  PROC DrawPart220()
    MoveL Offs(pOrigin,226.14,210.19,0.00),v60,z0,tPen\WObj:=wPaper;
    MoveL Offs(pOrigin,227.79,208.54,0.00),v40,fine,tPen\WObj:=wPaper;
    MoveL Offs(pOrigin,227.79,208.54,6.00),v60,z5,tPen\WObj:=wPaper;
    MoveL Offs(pOrigin,229.18,204.08,6.00),vTravel,z5,tPen\WObj:=wPaper;
    MoveL Offs(pOrigin,229.18,204.08,0.00),v60,z0,tPen\WObj:=wPaper;
    MoveL Offs(pOrigin,226.47,201.38,0.00),v40,fine,tPen\WObj:=wPaper;
    MoveL Offs(pOrigin,226.47,201.38,6.00),v60,z5,tPen\WObj:=wPaper;
    MoveL Offs(pOrigin,223.02,201.36,6.00),vTravel,z5,tPen\WObj:=wPaper;
    MoveL Offs(pOrigin,223.02,201.36,0.00),v60,z0,tPen\WObj:=wPaper;
    MoveL Offs(pOrigin,219.26,205.12,0.00),v40,fine,tPen\WObj:=wPaper;
    MoveL Offs(pOrigin,219.26,205.12,6.00),v60,z5,tPen\WObj:=wPaper;
    MoveL Offs(pOrigin,220.18,199.72,6.00),vTravel,z5,tPen\WObj:=wPaper;
    MoveL Offs(pOrigin,220.18,199.72,0.00),v60,z0,tPen\WObj:=wPaper;
    MoveL Offs(pOrigin,224.23,195.66,0.00),v40,fine,tPen\WObj:=wPaper;
    MoveL Offs(pOrigin,224.23,195.66,6.00),v60,z5,tPen\WObj:=wPaper;
    MoveL Offs(pOrigin,224.69,193.71,6.00),vTravel,z5,tPen\WObj:=wPaper;
    MoveL Offs(pOrigin,224.69,193.71,0.00),v60,z0,tPen\WObj:=wPaper;
    MoveL Offs(pOrigin,220.63,197.77,0.00),v40,fine,tPen\WObj:=wPaper;
    MoveL Offs(pOrigin,220.63,197.77,6.00),v60,z5,tPen\WObj:=wPaper;
    MoveL Offs(pOrigin,221.31,199.80,6.00),vTravel,z5,tPen\WObj:=wPaper;
    MoveL Offs(pOrigin,221.31,199.80,0.00),v60,z0,tPen\WObj:=wPaper;
    MoveL Offs(pOrigin,222.38,199.80,0.00),v40,fine,tPen\WObj:=wPaper;
    MoveL Offs(pOrigin,222.38,199.80,6.00),v60,z5,tPen\WObj:=wPaper;
    MoveL Offs(pOrigin,219.89,195.53,6.00),vTravel,z5,tPen\WObj:=wPaper;
    MoveL Offs(pOrigin,219.89,195.53,0.00),v60,z0,tPen\WObj:=wPaper;
    MoveL Offs(pOrigin,225.75,189.67,0.00),v40,fine,tPen\WObj:=wPaper;
    MoveL Offs(pOrigin,225.75,189.67,6.00),v60,z5,tPen\WObj:=wPaper;
    MoveL Offs(pOrigin,228.60,186.81,6.00),vTravel,z5,tPen\WObj:=wPaper;
    MoveL Offs(pOrigin,228.60,186.81,0.00),v60,z0,tPen\WObj:=wPaper;
    MoveL Offs(pOrigin,231.01,184.41,0.00),v40,z0,tPen\WObj:=wPaper;
    MoveL Offs(pOrigin,230.32,184.31,0.00),v40,z0,tPen\WObj:=wPaper;
    MoveL Offs(pOrigin,228.21,182.21,0.00),v40,fine,tPen\WObj:=wPaper;
    MoveL Offs(pOrigin,228.21,182.21,6.00),v60,z5,tPen\WObj:=wPaper;
    MoveL Offs(pOrigin,226.72,182.21,6.00),vTravel,z5,tPen\WObj:=wPaper;
    MoveL Offs(pOrigin,226.72,182.21,0.00),v60,z0,tPen\WObj:=wPaper;
    MoveL Offs(pOrigin,224.76,180.25,0.00),v40,z0,tPen\WObj:=wPaper;
    MoveL Offs(pOrigin,224.28,180.68,0.00),v40,z0,tPen\WObj:=wPaper;
    MoveL Offs(pOrigin,230.29,174.67,0.00),v40,z0,tPen\WObj:=wPaper;
    MoveL Offs(pOrigin,229.84,173.63,0.00),v40,z0,tPen\WObj:=wPaper;
    MoveL Offs(pOrigin,224.43,179.04,0.00),v40,z0,tPen\WObj:=wPaper;
    MoveL Offs(pOrigin,224.91,178.91,0.00),v40,z0,tPen\WObj:=wPaper;
    MoveL Offs(pOrigin,226.86,180.86,0.00),v40,z0,tPen\WObj:=wPaper;
    MoveL Offs(pOrigin,226.41,180.79,0.00),v40,z0,tPen\WObj:=wPaper;
    MoveL Offs(pOrigin,225.14,180.79,0.00),v40,z0,tPen\WObj:=wPaper;
    MoveL Offs(pOrigin,224.62,181.60,0.00),v40,z0,tPen\WObj:=wPaper;
    MoveL Offs(pOrigin,226.42,183.40,0.00),v40,z0,tPen\WObj:=wPaper;
    MoveL Offs(pOrigin,225.99,182.90,0.00),v40,z0,tPen\WObj:=wPaper;
    MoveL Offs(pOrigin,224.92,182.90,0.00),v40,z0,tPen\WObj:=wPaper;
    MoveL Offs(pOrigin,224.71,183.96,0.00),v40,z0,tPen\WObj:=wPaper;
    MoveL Offs(pOrigin,225.78,183.96,0.00),v40,fine,tPen\WObj:=wPaper;
    MoveL Offs(pOrigin,225.78,183.96,6.00),v60,z5,tPen\WObj:=wPaper;
    MoveL Offs(pOrigin,226.20,181.85,6.00),vTravel,z5,tPen\WObj:=wPaper;
    MoveL Offs(pOrigin,226.20,181.85,0.00),v60,z0,tPen\WObj:=wPaper;
    MoveL Offs(pOrigin,225.14,181.85,0.00),v40,fine,tPen\WObj:=wPaper;
    MoveL Offs(pOrigin,225.14,181.85,6.00),v60,z5,tPen\WObj:=wPaper;
    MoveL Offs(pOrigin,225.35,179.74,6.00),vTravel,z5,tPen\WObj:=wPaper;
    MoveL Offs(pOrigin,225.35,179.74,0.00),v60,z0,tPen\WObj:=wPaper;
    MoveL Offs(pOrigin,226.62,179.74,0.00),v40,z0,tPen\WObj:=wPaper;
    MoveL Offs(pOrigin,226.84,178.68,0.00),v40,z0,tPen\WObj:=wPaper;
    MoveL Offs(pOrigin,225.56,178.68,0.00),v40,fine,tPen\WObj:=wPaper;
    MoveL Offs(pOrigin,225.56,178.68,6.00),v60,z5,tPen\WObj:=wPaper;
    MoveL Offs(pOrigin,226.20,174.46,6.00),vTravel,z5,tPen\WObj:=wPaper;
    MoveL Offs(pOrigin,226.20,174.46,0.00),v60,z0,tPen\WObj:=wPaper;
    MoveL Offs(pOrigin,228.96,174.46,0.00),v40,fine,tPen\WObj:=wPaper;
    MoveL Offs(pOrigin,228.96,174.46,6.00),v60,z5,tPen\WObj:=wPaper;
    MoveL Offs(pOrigin,234.06,174.15,6.00),vTravel,z5,tPen\WObj:=wPaper;
    MoveL Offs(pOrigin,234.06,174.15,0.00),v60,z0,tPen\WObj:=wPaper;
    MoveL Offs(pOrigin,233.64,174.57,0.00),v40,z0,tPen\WObj:=wPaper;
    MoveL Offs(pOrigin,234.06,174.15,0.00),v40,fine,tPen\WObj:=wPaper;
    MoveL Offs(pOrigin,234.06,174.15,6.00),v60,z5,tPen\WObj:=wPaper;
    MoveL Offs(pOrigin,242.72,174.32,6.00),vTravel,z5,tPen\WObj:=wPaper;
    MoveL Offs(pOrigin,242.72,174.32,0.00),v60,z0,tPen\WObj:=wPaper;
    MoveL Offs(pOrigin,244.22,175.82,0.00),v40,fine,tPen\WObj:=wPaper;
    MoveL Offs(pOrigin,244.22,175.82,6.00),v60,z5,tPen\WObj:=wPaper;
    MoveL Offs(pOrigin,245.11,173.72,6.00),vTravel,z5,tPen\WObj:=wPaper;
    MoveL Offs(pOrigin,245.11,173.72,0.00),v60,z0,tPen\WObj:=wPaper;
    MoveL Offs(pOrigin,243.31,171.92,0.00),v40,fine,tPen\WObj:=wPaper;
    MoveL Offs(pOrigin,243.31,171.92,6.00),v60,z5,tPen\WObj:=wPaper;
    MoveL Offs(pOrigin,244.69,170.23,6.00),vTravel,z5,tPen\WObj:=wPaper;
    MoveL Offs(pOrigin,244.69,170.23,0.00),v60,z0,tPen\WObj:=wPaper;
    MoveL Offs(pOrigin,245.75,170.23,0.00),v40,z0,tPen\WObj:=wPaper;
    MoveL Offs(pOrigin,245.54,170.75,0.00),v40,z0,tPen\WObj:=wPaper;
    MoveL Offs(pOrigin,245.32,171.18,0.00),v40,z0,tPen\WObj:=wPaper;
    MoveL Offs(pOrigin,245.54,170.75,0.00),v40,z0,tPen\WObj:=wPaper;
    MoveL Offs(pOrigin,245.71,171.33,0.00),v40,z0,tPen\WObj:=wPaper;
    MoveL Offs(pOrigin,244.35,169.98,0.00),v40,z0,tPen\WObj:=wPaper;
    MoveL Offs(pOrigin,244.69,169.90,0.00),v40,z0,tPen\WObj:=wPaper;
    MoveL Offs(pOrigin,244.26,170.54,0.00),v40,z0,tPen\WObj:=wPaper;
    MoveL Offs(pOrigin,244.69,169.90,0.00),v40,z0,tPen\WObj:=wPaper;
    MoveL Offs(pOrigin,244.95,169.08,0.00),v40,z0,tPen\WObj:=wPaper;
    MoveL Offs(pOrigin,246.30,170.43,0.00),v40,z0,tPen\WObj:=wPaper;
    MoveL Offs(pOrigin,247.20,169.84,0.00),v40,z0,tPen\WObj:=wPaper;
    MoveL Offs(pOrigin,245.70,168.33,0.00),v40,z0,tPen\WObj:=wPaper;
    MoveL Offs(pOrigin,245.96,168.41,0.00),v40,z0,tPen\WObj:=wPaper;
    MoveL Offs(pOrigin,245.32,169.05,0.00),v40,z0,tPen\WObj:=wPaper;
    MoveL Offs(pOrigin,245.96,168.41,0.00),v40,z0,tPen\WObj:=wPaper;
    MoveL Offs(pOrigin,245.54,169.18,0.00),v40,z0,tPen\WObj:=wPaper;
    MoveL Offs(pOrigin,246.81,169.18,0.00),v40,z0,tPen\WObj:=wPaper;
    MoveL Offs(pOrigin,246.81,169.26,0.00),v40,z0,tPen\WObj:=wPaper;
    MoveL Offs(pOrigin,245.75,170.32,0.00),v40,z0,tPen\WObj:=wPaper;
    MoveL Offs(pOrigin,246.81,169.26,0.00),v40,fine,tPen\WObj:=wPaper;
    MoveL Offs(pOrigin,246.81,169.26,6.00),v60,z5,tPen\WObj:=wPaper;
    MoveL Offs(pOrigin,241.29,179.04,6.00),vTravel,z5,tPen\WObj:=wPaper;
    MoveL Offs(pOrigin,241.29,179.04,0.00),v60,z0,tPen\WObj:=wPaper;
    MoveL Offs(pOrigin,241.07,179.46,0.00),v40,z0,tPen\WObj:=wPaper;
    MoveL Offs(pOrigin,241.29,179.04,0.00),v40,z0,tPen\WObj:=wPaper;
    MoveL Offs(pOrigin,241.08,179.74,0.00),v40,z0,tPen\WObj:=wPaper;
    MoveL Offs(pOrigin,242.35,179.74,0.00),v40,fine,tPen\WObj:=wPaper;
    MoveL Offs(pOrigin,242.35,179.74,6.00),v60,z5,tPen\WObj:=wPaper;
    MoveL Offs(pOrigin,240.44,180.74,6.00),vTravel,z5,tPen\WObj:=wPaper;
    MoveL Offs(pOrigin,240.44,180.74,0.00),v60,z0,tPen\WObj:=wPaper;
    MoveL Offs(pOrigin,240.23,181.16,0.00),v40,z0,tPen\WObj:=wPaper;
    MoveL Offs(pOrigin,240.44,180.74,0.00),v40,fine,tPen\WObj:=wPaper;
    MoveL Offs(pOrigin,240.44,180.74,6.00),v60,z5,tPen\WObj:=wPaper;
    MoveL Offs(pOrigin,241.29,181.80,6.00),vTravel,z5,tPen\WObj:=wPaper;
    MoveL Offs(pOrigin,241.29,181.80,0.00),v60,z0,tPen\WObj:=wPaper;
    MoveL Offs(pOrigin,240.86,182.44,0.00),v40,z0,tPen\WObj:=wPaper;
    MoveL Offs(pOrigin,241.29,181.80,0.00),v40,fine,tPen\WObj:=wPaper;
    MoveL Offs(pOrigin,241.29,181.80,6.00),v60,z5,tPen\WObj:=wPaper;
    MoveL Offs(pOrigin,243.12,190.21,6.00),vTravel,z5,tPen\WObj:=wPaper;
  ENDPROC

  PROC DrawPart221()
    MoveL Offs(pOrigin,243.12,190.21,0.00),v60,z0,tPen\WObj:=wPaper;
    MoveL Offs(pOrigin,241.02,192.32,0.00),v40,fine,tPen\WObj:=wPaper;
    MoveL Offs(pOrigin,241.02,192.32,6.00),v60,z5,tPen\WObj:=wPaper;
    MoveL Offs(pOrigin,242.97,191.86,6.00),vTravel,z5,tPen\WObj:=wPaper;
    MoveL Offs(pOrigin,242.97,191.86,0.00),v60,z0,tPen\WObj:=wPaper;
    MoveL Offs(pOrigin,244.47,190.36,0.00),v40,fine,tPen\WObj:=wPaper;
    MoveL Offs(pOrigin,244.47,190.36,6.00),v60,z5,tPen\WObj:=wPaper;
    MoveL Offs(pOrigin,244.77,191.56,6.00),vTravel,z5,tPen\WObj:=wPaper;
    MoveL Offs(pOrigin,244.77,191.56,0.00),v60,z0,tPen\WObj:=wPaper;
    MoveL Offs(pOrigin,245.82,190.50,0.00),v40,fine,tPen\WObj:=wPaper;
    MoveL Offs(pOrigin,245.82,190.50,6.00),v60,z5,tPen\WObj:=wPaper;
    MoveL Offs(pOrigin,251.66,192.13,6.00),vTravel,z5,tPen\WObj:=wPaper;
    MoveL Offs(pOrigin,251.66,192.13,0.00),v60,z0,tPen\WObj:=wPaper;
    MoveL Offs(pOrigin,252.56,191.23,0.00),v40,fine,tPen\WObj:=wPaper;
    MoveL Offs(pOrigin,252.56,191.23,6.00),v60,z5,tPen\WObj:=wPaper;
    MoveL Offs(pOrigin,252.85,192.43,6.00),vTravel,z5,tPen\WObj:=wPaper;
    MoveL Offs(pOrigin,252.85,192.43,0.00),v60,z0,tPen\WObj:=wPaper;
    MoveL Offs(pOrigin,254.81,190.48,0.00),v40,fine,tPen\WObj:=wPaper;
    MoveL Offs(pOrigin,254.81,190.48,6.00),v60,z5,tPen\WObj:=wPaper;
    MoveL Offs(pOrigin,254.50,192.28,6.00),vTravel,z5,tPen\WObj:=wPaper;
    MoveL Offs(pOrigin,254.50,192.28,0.00),v60,z0,tPen\WObj:=wPaper;
    MoveL Offs(pOrigin,256.76,190.02,0.00),v40,fine,tPen\WObj:=wPaper;
    MoveL Offs(pOrigin,256.76,190.02,6.00),v60,z5,tPen\WObj:=wPaper;
    MoveL Offs(pOrigin,258.26,190.02,6.00),vTravel,z5,tPen\WObj:=wPaper;
    MoveL Offs(pOrigin,258.26,190.02,0.00),v60,z0,tPen\WObj:=wPaper;
    MoveL Offs(pOrigin,256.30,191.97,0.00),v40,fine,tPen\WObj:=wPaper;
    MoveL Offs(pOrigin,256.30,191.97,6.00),v60,z5,tPen\WObj:=wPaper;
    MoveL Offs(pOrigin,257.80,191.97,6.00),vTravel,z5,tPen\WObj:=wPaper;
    MoveL Offs(pOrigin,257.80,191.97,0.00),v60,z0,tPen\WObj:=wPaper;
    MoveL Offs(pOrigin,259.75,190.01,0.00),v40,fine,tPen\WObj:=wPaper;
    MoveL Offs(pOrigin,259.75,190.01,6.00),v60,z5,tPen\WObj:=wPaper;
    MoveL Offs(pOrigin,260.95,190.31,6.00),vTravel,z5,tPen\WObj:=wPaper;
    MoveL Offs(pOrigin,260.95,190.31,0.00),v60,z0,tPen\WObj:=wPaper;
    MoveL Offs(pOrigin,259.30,191.96,0.00),v40,fine,tPen\WObj:=wPaper;
    MoveL Offs(pOrigin,259.30,191.96,6.00),v60,z5,tPen\WObj:=wPaper;
    MoveL Offs(pOrigin,260.80,191.96,6.00),vTravel,z5,tPen\WObj:=wPaper;
    MoveL Offs(pOrigin,260.80,191.96,0.00),v60,z0,tPen\WObj:=wPaper;
    MoveL Offs(pOrigin,262.30,190.45,0.00),v40,z0,tPen\WObj:=wPaper;
    MoveL Offs(pOrigin,262.85,191.46,0.00),v40,z0,tPen\WObj:=wPaper;
    MoveL Offs(pOrigin,263.90,192.51,0.00),v40,z0,tPen\WObj:=wPaper;
    MoveL Offs(pOrigin,263.04,192.70,0.00),v40,z0,tPen\WObj:=wPaper;
    MoveL Offs(pOrigin,264.69,191.05,0.00),v40,z0,tPen\WObj:=wPaper;
    MoveL Offs(pOrigin,263.65,190.60,0.00),v40,z0,tPen\WObj:=wPaper;
    MoveL Offs(pOrigin,261.84,192.40,0.00),v40,fine,tPen\WObj:=wPaper;
    MoveL Offs(pOrigin,261.84,192.40,6.00),v60,z5,tPen\WObj:=wPaper;
    MoveL Offs(pOrigin,256.70,208.00,6.00),vTravel,z5,tPen\WObj:=wPaper;
    MoveL Offs(pOrigin,256.70,208.00,0.00),v60,z0,tPen\WObj:=wPaper;
    MoveL Offs(pOrigin,254.45,210.25,0.00),v40,z0,tPen\WObj:=wPaper;
    MoveL Offs(pOrigin,254.51,210.00,0.00),v40,z0,tPen\WObj:=wPaper;
    MoveL Offs(pOrigin,252.41,207.90,0.00),v40,z0,tPen\WObj:=wPaper;
    MoveL Offs(pOrigin,251.70,208.25,0.00),v40,z0,tPen\WObj:=wPaper;
    MoveL Offs(pOrigin,248.94,208.25,0.00),v40,fine,tPen\WObj:=wPaper;
    MoveL Offs(pOrigin,248.94,208.25,6.00),v60,z5,tPen\WObj:=wPaper;
    MoveL Offs(pOrigin,250.40,209.81,6.00),vTravel,z5,tPen\WObj:=wPaper;
    MoveL Offs(pOrigin,250.40,209.81,0.00),v60,z0,tPen\WObj:=wPaper;
    MoveL Offs(pOrigin,252.96,207.26,0.00),v40,fine,tPen\WObj:=wPaper;
    MoveL Offs(pOrigin,252.96,207.26,6.00),v60,z5,tPen\WObj:=wPaper;
    MoveL Offs(pOrigin,256.84,210.84,6.00),vTravel,z5,tPen\WObj:=wPaper;
    MoveL Offs(pOrigin,256.84,210.84,0.00),v60,z0,tPen\WObj:=wPaper;
    MoveL Offs(pOrigin,258.95,208.74,0.00),v40,fine,tPen\WObj:=wPaper;
    MoveL Offs(pOrigin,258.95,208.74,6.00),v60,z5,tPen\WObj:=wPaper;
    MoveL Offs(pOrigin,266.86,215.76,6.00),vTravel,z5,tPen\WObj:=wPaper;
    MoveL Offs(pOrigin,266.86,215.76,0.00),v60,z0,tPen\WObj:=wPaper;
    MoveL Offs(pOrigin,267.92,214.70,0.00),v40,fine,tPen\WObj:=wPaper;
    MoveL Offs(pOrigin,267.92,214.70,6.00),v60,z5,tPen\WObj:=wPaper;
    MoveL Offs(pOrigin,278.83,220.21,6.00),vTravel,z5,tPen\WObj:=wPaper;
    MoveL Offs(pOrigin,278.83,220.21,0.00),v60,z0,tPen\WObj:=wPaper;
    MoveL Offs(pOrigin,279.74,219.31,0.00),v40,z0,tPen\WObj:=wPaper;
    MoveL Offs(pOrigin,280.33,220.21,0.00),v40,z0,tPen\WObj:=wPaper;
    MoveL Offs(pOrigin,279.58,220.96,0.00),v40,fine,tPen\WObj:=wPaper;
    MoveL Offs(pOrigin,279.58,220.96,6.00),v60,z5,tPen\WObj:=wPaper;
    MoveL Offs(pOrigin,269.06,231.48,6.00),vTravel,z5,tPen\WObj:=wPaper;
    MoveL Offs(pOrigin,269.06,231.48,0.00),v60,z0,tPen\WObj:=wPaper;
    MoveL Offs(pOrigin,257.94,242.60,0.00),v40,z0,tPen\WObj:=wPaper;
    MoveL Offs(pOrigin,258.21,242.07,0.00),v40,z0,tPen\WObj:=wPaper;
    MoveL Offs(pOrigin,250.69,234.56,0.00),v40,z0,tPen\WObj:=wPaper;
    MoveL Offs(pOrigin,250.64,235.35,0.00),v40,z0,tPen\WObj:=wPaper;
    MoveL Offs(pOrigin,251.27,234.93,0.00),v40,z0,tPen\WObj:=wPaper;
    MoveL Offs(pOrigin,252.55,234.93,0.00),v40,z0,tPen\WObj:=wPaper;
    MoveL Offs(pOrigin,252.98,235.35,0.00),v40,z0,tPen\WObj:=wPaper;
    MoveL Offs(pOrigin,252.98,235.35,0.00),v40,z0,tPen\WObj:=wPaper;
    MoveL Offs(pOrigin,254.04,235.14,0.00),v40,z0,tPen\WObj:=wPaper;
    MoveL Offs(pOrigin,254.46,235.56,0.00),v40,z0,tPen\WObj:=wPaper;
    MoveL Offs(pOrigin,254.46,235.56,0.00),v40,z0,tPen\WObj:=wPaper;
    MoveL Offs(pOrigin,254.04,235.99,0.00),v40,z0,tPen\WObj:=wPaper;
    MoveL Offs(pOrigin,252.98,235.99,0.00),v40,z0,tPen\WObj:=wPaper;
    MoveL Offs(pOrigin,252.98,235.99,0.00),v40,z0,tPen\WObj:=wPaper;
    MoveL Offs(pOrigin,251.49,236.20,0.00),v40,z0,tPen\WObj:=wPaper;
    MoveL Offs(pOrigin,251.34,235.99,0.00),v40,z0,tPen\WObj:=wPaper;
    MoveL Offs(pOrigin,251.34,241.51,0.00),v40,z0,tPen\WObj:=wPaper;
    MoveL Offs(pOrigin,250.29,241.51,0.00),v40,z0,tPen\WObj:=wPaper;
    MoveL Offs(pOrigin,250.29,235.99,0.00),v40,z0,tPen\WObj:=wPaper;
    MoveL Offs(pOrigin,250.64,235.35,0.00),v40,z0,tPen\WObj:=wPaper;
    MoveL Offs(pOrigin,249.36,235.35,0.00),v40,z0,tPen\WObj:=wPaper;
    MoveL Offs(pOrigin,249.36,235.35,0.00),v40,z0,tPen\WObj:=wPaper;
    MoveL Offs(pOrigin,248.73,234.93,0.00),v40,z0,tPen\WObj:=wPaper;
    MoveL Offs(pOrigin,247.24,234.78,0.00),v40,z0,tPen\WObj:=wPaper;
    MoveL Offs(pOrigin,247.45,235.99,0.00),v40,z0,tPen\WObj:=wPaper;
    MoveL Offs(pOrigin,247.02,236.62,0.00),v40,z0,tPen\WObj:=wPaper;
    MoveL Offs(pOrigin,247.12,235.99,0.00),v40,z0,tPen\WObj:=wPaper;
    MoveL Offs(pOrigin,247.12,239.81,0.00),v40,z0,tPen\WObj:=wPaper;
    MoveL Offs(pOrigin,246.18,239.93,0.00),v40,z0,tPen\WObj:=wPaper;
    MoveL Offs(pOrigin,267.85,239.93,0.00),v40,z0,tPen\WObj:=wPaper;
    MoveL Offs(pOrigin,267.18,239.39,0.00),v40,z0,tPen\WObj:=wPaper;
    MoveL Offs(pOrigin,267.18,232.80,0.00),v40,z0,tPen\WObj:=wPaper;
    MoveL Offs(pOrigin,267.00,231.95,0.00),v40,z0,tPen\WObj:=wPaper;
    MoveL Offs(pOrigin,268.06,231.95,0.00),v40,z0,tPen\WObj:=wPaper;
    MoveL Offs(pOrigin,268.06,231.95,0.00),v40,z0,tPen\WObj:=wPaper;
    MoveL Offs(pOrigin,268.06,231.10,0.00),v40,z0,tPen\WObj:=wPaper;
    MoveL Offs(pOrigin,267.64,230.68,0.00),v40,z0,tPen\WObj:=wPaper;
    MoveL Offs(pOrigin,267.64,230.68,0.00),v40,z0,tPen\WObj:=wPaper;
    MoveL Offs(pOrigin,267.00,231.95,0.00),v40,z0,tPen\WObj:=wPaper;
    MoveL Offs(pOrigin,267.00,231.95,0.00),v40,z0,tPen\WObj:=wPaper;
    MoveL Offs(pOrigin,265.51,232.52,0.00),v40,z0,tPen\WObj:=wPaper;
    MoveL Offs(pOrigin,264.88,233.44,0.00),v40,z0,tPen\WObj:=wPaper;
    MoveL Offs(pOrigin,262.96,233.65,0.00),v40,z0,tPen\WObj:=wPaper;
    MoveL Offs(pOrigin,259.35,232.73,0.00),v40,z0,tPen\WObj:=wPaper;
    MoveL Offs(pOrigin,258.43,231.31,0.00),v40,z0,tPen\WObj:=wPaper;
    MoveL Offs(pOrigin,257.44,230.60,0.00),v40,z0,tPen\WObj:=wPaper;
    MoveL Offs(pOrigin,251.91,228.34,0.00),v40,z0,tPen\WObj:=wPaper;
  ENDPROC

  PROC DrawPart222()
    MoveL Offs(pOrigin,243.62,227.06,0.00),v40,z0,tPen\WObj:=wPaper;
    MoveL Offs(pOrigin,239.80,227.06,0.00),v40,z0,tPen\WObj:=wPaper;
    MoveL Offs(pOrigin,237.25,227.49,0.00),v40,fine,tPen\WObj:=wPaper;
    MoveL Offs(pOrigin,237.25,227.49,6.00),v60,z5,tPen\WObj:=wPaper;
    MoveL Offs(pOrigin,235.82,228.88,6.00),vTravel,z5,tPen\WObj:=wPaper;
    MoveL Offs(pOrigin,235.82,228.88,0.00),v60,z0,tPen\WObj:=wPaper;
    MoveL Offs(pOrigin,225.75,238.95,0.00),v40,z0,tPen\WObj:=wPaper;
    MoveL Offs(pOrigin,225.00,238.20,0.00),v40,z0,tPen\WObj:=wPaper;
    MoveL Offs(pOrigin,234.77,228.44,0.00),v40,fine,tPen\WObj:=wPaper;
    MoveL Offs(pOrigin,234.77,228.44,6.00),v60,z5,tPen\WObj:=wPaper;
    MoveL Offs(pOrigin,233.27,228.44,6.00),vTravel,z5,tPen\WObj:=wPaper;
    MoveL Offs(pOrigin,233.27,228.44,0.00),v60,z0,tPen\WObj:=wPaper;
    MoveL Offs(pOrigin,224.41,237.31,0.00),v40,z0,tPen\WObj:=wPaper;
    MoveL Offs(pOrigin,223.81,236.41,0.00),v40,z0,tPen\WObj:=wPaper;
    MoveL Offs(pOrigin,231.77,228.45,0.00),v40,z0,tPen\WObj:=wPaper;
    MoveL Offs(pOrigin,231.80,229.11,0.00),v40,z0,tPen\WObj:=wPaper;
    MoveL Offs(pOrigin,242.77,240.08,0.00),v40,z0,tPen\WObj:=wPaper;
    MoveL Offs(pOrigin,243.72,240.39,0.00),v40,z0,tPen\WObj:=wPaper;
    MoveL Offs(pOrigin,252.28,231.83,0.00),v40,z0,tPen\WObj:=wPaper;
    MoveL Offs(pOrigin,251.74,232.62,0.00),v40,z0,tPen\WObj:=wPaper;
    MoveL Offs(pOrigin,260.75,241.63,0.00),v40,z0,tPen\WObj:=wPaper;
    MoveL Offs(pOrigin,260.84,240.88,0.00),v40,z0,tPen\WObj:=wPaper;
    MoveL Offs(pOrigin,262.54,241.16,0.00),v40,z0,tPen\WObj:=wPaper;
    MoveL Offs(pOrigin,263.39,240.88,0.00),v40,z0,tPen\WObj:=wPaper;
    MoveL Offs(pOrigin,263.45,241.34,0.00),v40,z0,tPen\WObj:=wPaper;
    MoveL Offs(pOrigin,255.18,233.08,0.00),v40,z0,tPen\WObj:=wPaper;
    MoveL Offs(pOrigin,255.13,231.97,0.00),v40,z0,tPen\WObj:=wPaper;
    MoveL Offs(pOrigin,245.81,241.29,0.00),v40,z0,tPen\WObj:=wPaper;
    MoveL Offs(pOrigin,246.41,242.18,0.00),v40,z0,tPen\WObj:=wPaper;
    MoveL Offs(pOrigin,256.63,231.97,0.00),v40,z0,tPen\WObj:=wPaper;
    MoveL Offs(pOrigin,256.68,233.08,0.00),v40,z0,tPen\WObj:=wPaper;
    MoveL Offs(pOrigin,265.25,241.65,0.00),v40,fine,tPen\WObj:=wPaper;
    MoveL Offs(pOrigin,265.25,241.65,6.00),v60,z5,tPen\WObj:=wPaper;
    MoveL Offs(pOrigin,266.36,240.66,6.00),vTravel,z5,tPen\WObj:=wPaper;
    MoveL Offs(pOrigin,266.36,240.66,0.00),v60,z0,tPen\WObj:=wPaper;
    MoveL Offs(pOrigin,265.73,242.57,0.00),v40,z0,tPen\WObj:=wPaper;
    MoveL Offs(pOrigin,264.02,244.06,0.00),v40,z0,tPen\WObj:=wPaper;
    MoveL Offs(pOrigin,263.60,244.27,0.00),v40,z0,tPen\WObj:=wPaper;
    MoveL Offs(pOrigin,257.23,249.80,0.00),v40,z0,tPen\WObj:=wPaper;
    MoveL Offs(pOrigin,255.74,250.23,0.00),v40,z0,tPen\WObj:=wPaper;
    MoveL Offs(pOrigin,255.74,250.23,0.00),v40,z0,tPen\WObj:=wPaper;
    MoveL Offs(pOrigin,254.46,251.29,0.00),v40,z0,tPen\WObj:=wPaper;
    MoveL Offs(pOrigin,254.39,251.36,0.00),v40,z0,tPen\WObj:=wPaper;
    MoveL Offs(pOrigin,254.04,252.07,0.00),v40,z0,tPen\WObj:=wPaper;
    MoveL Offs(pOrigin,253.47,252.14,0.00),v40,z0,tPen\WObj:=wPaper;
    MoveL Offs(pOrigin,253.61,251.36,0.00),v40,z0,tPen\WObj:=wPaper;
    MoveL Offs(pOrigin,254.39,251.36,0.00),v40,z0,tPen\WObj:=wPaper;
    MoveL Offs(pOrigin,254.62,251.90,0.00),v40,z0,tPen\WObj:=wPaper;
    MoveL Offs(pOrigin,262.28,244.23,0.00),v40,fine,tPen\WObj:=wPaper;
    MoveL Offs(pOrigin,262.28,244.23,6.00),v60,z5,tPen\WObj:=wPaper;
    MoveL Offs(pOrigin,261.39,242.14,6.00),vTravel,z5,tPen\WObj:=wPaper;
    MoveL Offs(pOrigin,261.39,242.14,0.00),v60,z0,tPen\WObj:=wPaper;
    MoveL Offs(pOrigin,270.41,233.12,0.00),v40,z0,tPen\WObj:=wPaper;
    MoveL Offs(pOrigin,269.55,233.59,0.00),v40,z0,tPen\WObj:=wPaper;
    MoveL Offs(pOrigin,259.35,233.59,0.00),v40,z0,tPen\WObj:=wPaper;
    MoveL Offs(pOrigin,259.14,233.23,0.00),v40,z0,tPen\WObj:=wPaper;
    MoveL Offs(pOrigin,258.50,233.65,0.00),v40,z0,tPen\WObj:=wPaper;
    MoveL Offs(pOrigin,254.25,233.44,0.00),v40,z0,tPen\WObj:=wPaper;
    MoveL Offs(pOrigin,248.09,232.16,0.00),v40,z0,tPen\WObj:=wPaper;
    MoveL Offs(pOrigin,245.54,231.95,0.00),v40,z0,tPen\WObj:=wPaper;
    MoveL Offs(pOrigin,245.54,231.95,0.00),v40,z0,tPen\WObj:=wPaper;
    MoveL Offs(pOrigin,245.11,231.31,0.00),v40,z0,tPen\WObj:=wPaper;
    MoveL Offs(pOrigin,244.48,231.31,0.00),v40,z0,tPen\WObj:=wPaper;
    MoveL Offs(pOrigin,244.26,231.74,0.00),v40,z0,tPen\WObj:=wPaper;
    MoveL Offs(pOrigin,244.26,231.74,0.00),v40,z0,tPen\WObj:=wPaper;
    MoveL Offs(pOrigin,244.69,232.16,0.00),v40,z0,tPen\WObj:=wPaper;
    MoveL Offs(pOrigin,245.54,231.95,0.00),v40,z0,tPen\WObj:=wPaper;
    MoveL Offs(pOrigin,245.74,232.60,0.00),v40,z0,tPen\WObj:=wPaper;
    MoveL Offs(pOrigin,244.54,231.40,0.00),v40,z0,tPen\WObj:=wPaper;
    MoveL Offs(pOrigin,244.26,231.74,0.00),v40,z0,tPen\WObj:=wPaper;
    MoveL Offs(pOrigin,240.65,231.74,0.00),v40,z0,tPen\WObj:=wPaper;
    MoveL Offs(pOrigin,234.70,230.68,0.00),v40,z0,tPen\WObj:=wPaper;
    MoveL Offs(pOrigin,234.70,230.68,0.00),v40,z0,tPen\WObj:=wPaper;
    MoveL Offs(pOrigin,234.06,229.82,0.00),v40,z0,tPen\WObj:=wPaper;
    MoveL Offs(pOrigin,233.21,229.40,0.00),v40,z0,tPen\WObj:=wPaper;
    MoveL Offs(pOrigin,231.09,229.75,0.00),v40,z0,tPen\WObj:=wPaper;
    MoveL Offs(pOrigin,230.45,229.05,0.00),v40,z0,tPen\WObj:=wPaper;
    MoveL Offs(pOrigin,228.75,228.20,0.00),v40,z0,tPen\WObj:=wPaper;
    MoveL Offs(pOrigin,228.32,227.35,0.00),v40,z0,tPen\WObj:=wPaper;
    MoveL Offs(pOrigin,227.05,226.64,0.00),v40,z0,tPen\WObj:=wPaper;
    MoveL Offs(pOrigin,225.77,226.99,0.00),v40,z0,tPen\WObj:=wPaper;
    MoveL Offs(pOrigin,223.65,228.55,0.00),v40,z0,tPen\WObj:=wPaper;
    MoveL Offs(pOrigin,223.23,230.25,0.00),v40,z0,tPen\WObj:=wPaper;
    MoveL Offs(pOrigin,223.23,230.25,0.00),v40,z0,tPen\WObj:=wPaper;
    MoveL Offs(pOrigin,224.07,230.89,0.00),v40,z0,tPen\WObj:=wPaper;
    MoveL Offs(pOrigin,223.86,231.74,0.00),v40,z0,tPen\WObj:=wPaper;
    MoveL Offs(pOrigin,223.23,231.74,0.00),v40,z0,tPen\WObj:=wPaper;
    MoveL Offs(pOrigin,223.22,231.48,0.00),v40,z0,tPen\WObj:=wPaper;
    MoveL Offs(pOrigin,233.85,231.48,0.00),v40,z0,tPen\WObj:=wPaper;
    MoveL Offs(pOrigin,234.06,231.52,0.00),v40,z0,tPen\WObj:=wPaper;
    MoveL Offs(pOrigin,233.85,231.31,0.00),v40,z0,tPen\WObj:=wPaper;
    MoveL Offs(pOrigin,232.15,231.52,0.00),v40,z0,tPen\WObj:=wPaper;
    MoveL Offs(pOrigin,232.15,231.52,0.00),v40,z0,tPen\WObj:=wPaper;
    MoveL Offs(pOrigin,232.79,232.38,0.00),v40,z0,tPen\WObj:=wPaper;
    MoveL Offs(pOrigin,234.06,232.16,0.00),v40,z0,tPen\WObj:=wPaper;
    MoveL Offs(pOrigin,234.06,232.16,0.00),v40,z0,tPen\WObj:=wPaper;
    MoveL Offs(pOrigin,234.70,233.23,0.00),v40,z0,tPen\WObj:=wPaper;
    MoveL Offs(pOrigin,235.76,233.23,0.00),v40,z0,tPen\WObj:=wPaper;
    MoveL Offs(pOrigin,235.76,233.23,0.00),v40,z0,tPen\WObj:=wPaper;
    MoveL Offs(pOrigin,236.19,232.59,0.00),v40,z0,tPen\WObj:=wPaper;
    MoveL Offs(pOrigin,237.25,232.80,0.00),v40,z0,tPen\WObj:=wPaper;
    MoveL Offs(pOrigin,237.68,233.23,0.00),v40,z0,tPen\WObj:=wPaper;
    MoveL Offs(pOrigin,237.68,233.23,0.00),v40,z0,tPen\WObj:=wPaper;
    MoveL Offs(pOrigin,239.80,233.51,0.00),v40,z0,tPen\WObj:=wPaper;
    MoveL Offs(pOrigin,240.44,234.29,0.00),v40,z0,tPen\WObj:=wPaper;
    MoveL Offs(pOrigin,240.44,234.29,0.00),v40,z0,tPen\WObj:=wPaper;
    MoveL Offs(pOrigin,239.59,234.71,0.00),v40,z0,tPen\WObj:=wPaper;
    MoveL Offs(pOrigin,237.68,233.86,0.00),v40,z0,tPen\WObj:=wPaper;
    MoveL Offs(pOrigin,237.61,234.29,0.00),v40,z0,tPen\WObj:=wPaper;
    MoveL Offs(pOrigin,237.61,239.60,0.00),v40,z0,tPen\WObj:=wPaper;
    MoveL Offs(pOrigin,238.31,240.24,0.00),v40,z0,tPen\WObj:=wPaper;
    MoveL Offs(pOrigin,239.16,240.66,0.00),v40,z0,tPen\WObj:=wPaper;
    MoveL Offs(pOrigin,239.16,240.66,0.00),v40,z0,tPen\WObj:=wPaper;
    MoveL Offs(pOrigin,239.16,241.73,0.00),v40,z0,tPen\WObj:=wPaper;
    MoveL Offs(pOrigin,239.16,241.73,0.00),v40,z0,tPen\WObj:=wPaper;
    MoveL Offs(pOrigin,239.38,242.15,0.00),v40,z0,tPen\WObj:=wPaper;
    MoveL Offs(pOrigin,239.16,242.79,0.00),v40,z0,tPen\WObj:=wPaper;
    MoveL Offs(pOrigin,238.31,243.00,0.00),v40,z0,tPen\WObj:=wPaper;
    MoveL Offs(pOrigin,238.31,243.00,0.00),v40,z0,tPen\WObj:=wPaper;
    MoveL Offs(pOrigin,237.04,245.98,0.00),v40,z0,tPen\WObj:=wPaper;
  ENDPROC

  PROC DrawPart223()
    MoveL Offs(pOrigin,236.82,248.31,0.00),v40,fine,tPen\WObj:=wPaper;
    MoveL Offs(pOrigin,236.82,248.31,6.00),v60,z5,tPen\WObj:=wPaper;
    MoveL Offs(pOrigin,233.64,248.95,6.00),vTravel,z5,tPen\WObj:=wPaper;
    MoveL Offs(pOrigin,233.64,248.95,0.00),v60,z0,tPen\WObj:=wPaper;
    MoveL Offs(pOrigin,232.93,248.31,0.00),v40,z0,tPen\WObj:=wPaper;
    MoveL Offs(pOrigin,231.73,246.19,0.00),v40,z0,tPen\WObj:=wPaper;
    MoveL Offs(pOrigin,231.73,246.19,0.00),v40,z0,tPen\WObj:=wPaper;
    MoveL Offs(pOrigin,230.66,245.55,0.00),v40,z0,tPen\WObj:=wPaper;
    MoveL Offs(pOrigin,224.85,236.20,0.00),v40,z0,tPen\WObj:=wPaper;
    MoveL Offs(pOrigin,221.95,232.16,0.00),v40,z0,tPen\WObj:=wPaper;
    MoveL Offs(pOrigin,221.87,232.37,0.00),v40,z0,tPen\WObj:=wPaper;
    MoveL Offs(pOrigin,228.33,225.91,0.00),v40,z0,tPen\WObj:=wPaper;
    MoveL Offs(pOrigin,227.60,226.40,0.00),v40,z0,tPen\WObj:=wPaper;
    MoveL Offs(pOrigin,241.72,240.52,0.00),v40,z0,tPen\WObj:=wPaper;
    MoveL Offs(pOrigin,241.77,240.85,0.00),v40,z0,tPen\WObj:=wPaper;
    MoveL Offs(pOrigin,251.09,231.53,0.00),v40,fine,tPen\WObj:=wPaper;
    MoveL Offs(pOrigin,251.09,231.53,6.00),v60,z5,tPen\WObj:=wPaper;
    MoveL Offs(pOrigin,249.74,231.39,6.00),vTravel,z5,tPen\WObj:=wPaper;
    MoveL Offs(pOrigin,249.74,231.39,0.00),v60,z0,tPen\WObj:=wPaper;
    MoveL Offs(pOrigin,237.42,243.71,0.00),v40,z0,tPen\WObj:=wPaper;
    MoveL Offs(pOrigin,237.99,242.76,0.00),v40,z0,tPen\WObj:=wPaper;
    MoveL Offs(pOrigin,223.41,228.18,0.00),v40,z0,tPen\WObj:=wPaper;
    MoveL Offs(pOrigin,222.78,228.47,0.00),v40,z0,tPen\WObj:=wPaper;
    MoveL Offs(pOrigin,225.04,226.22,0.00),v40,z0,tPen\WObj:=wPaper;
    MoveL Offs(pOrigin,225.06,226.84,0.00),v40,z0,tPen\WObj:=wPaper;
    MoveL Offs(pOrigin,239.78,241.57,0.00),v40,z0,tPen\WObj:=wPaper;
    MoveL Offs(pOrigin,239.16,241.73,0.00),v40,z0,tPen\WObj:=wPaper;
    MoveL Offs(pOrigin,238.31,241.94,0.00),v40,z0,tPen\WObj:=wPaper;
    MoveL Offs(pOrigin,238.10,242.36,0.00),v40,z0,tPen\WObj:=wPaper;
    MoveL Offs(pOrigin,238.10,242.36,0.00),v40,z0,tPen\WObj:=wPaper;
    MoveL Offs(pOrigin,236.19,242.57,0.00),v40,z0,tPen\WObj:=wPaper;
    MoveL Offs(pOrigin,233.85,241.58,0.00),v40,z0,tPen\WObj:=wPaper;
    MoveL Offs(pOrigin,232.43,243.00,0.00),v40,z0,tPen\WObj:=wPaper;
    MoveL Offs(pOrigin,231.73,246.19,0.00),v40,z0,tPen\WObj:=wPaper;
    MoveL Offs(pOrigin,232.30,246.04,0.00),v40,z0,tPen\WObj:=wPaper;
    MoveL Offs(pOrigin,231.40,245.14,0.00),v40,fine,tPen\WObj:=wPaper;
    MoveL Offs(pOrigin,231.40,245.14,6.00),v60,z5,tPen\WObj:=wPaper;
    MoveL Offs(pOrigin,231.11,246.33,6.00),vTravel,z5,tPen\WObj:=wPaper;
    MoveL Offs(pOrigin,231.11,246.33,0.00),v60,z0,tPen\WObj:=wPaper;
    MoveL Offs(pOrigin,232.31,247.54,0.00),v40,z0,tPen\WObj:=wPaper;
    MoveL Offs(pOrigin,231.56,248.07,0.00),v40,z0,tPen\WObj:=wPaper;
    MoveL Offs(pOrigin,233.37,246.27,0.00),v40,z0,tPen\WObj:=wPaper;
    MoveL Offs(pOrigin,232.92,245.22,0.00),v40,z0,tPen\WObj:=wPaper;
    MoveL Offs(pOrigin,230.97,247.17,0.00),v40,z0,tPen\WObj:=wPaper;
    MoveL Offs(pOrigin,230.37,246.28,0.00),v40,z0,tPen\WObj:=wPaper;
    MoveL Offs(pOrigin,246.15,230.50,0.00),v40,z0,tPen\WObj:=wPaper;
    MoveL Offs(pOrigin,246.04,231.40,0.00),v40,z0,tPen\WObj:=wPaper;
    MoveL Offs(pOrigin,247.24,232.60,0.00),v40,z0,tPen\WObj:=wPaper;
    MoveL Offs(pOrigin,247.84,231.71,0.00),v40,z0,tPen\WObj:=wPaper;
    MoveL Offs(pOrigin,249.04,232.91,0.00),v40,z0,tPen\WObj:=wPaper;
    MoveL Offs(pOrigin,250.09,232.46,0.00),v40,z0,tPen\WObj:=wPaper;
    MoveL Offs(pOrigin,259.40,241.78,0.00),v40,z0,tPen\WObj:=wPaper;
    MoveL Offs(pOrigin,259.59,242.44,0.00),v40,z0,tPen\WObj:=wPaper;
    MoveL Offs(pOrigin,269.81,232.22,0.00),v40,fine,tPen\WObj:=wPaper;
    MoveL Offs(pOrigin,269.81,232.22,6.00),v60,z5,tPen\WObj:=wPaper;
    MoveL Offs(pOrigin,268.49,232.54,6.00),vTravel,z5,tPen\WObj:=wPaper;
    MoveL Offs(pOrigin,268.49,232.54,0.00),v60,z0,tPen\WObj:=wPaper;
    MoveL Offs(pOrigin,265.73,232.54,0.00),v40,z0,tPen\WObj:=wPaper;
    MoveL Offs(pOrigin,265.07,232.51,0.00),v40,z0,tPen\WObj:=wPaper;
    MoveL Offs(pOrigin,270.18,237.62,0.00),v40,z0,tPen\WObj:=wPaper;
    MoveL Offs(pOrigin,269.55,237.82,0.00),v40,z0,tPen\WObj:=wPaper;
    MoveL Offs(pOrigin,231.72,237.82,0.00),v40,z0,tPen\WObj:=wPaper;
    MoveL Offs(pOrigin,231.73,238.11,0.00),v40,z0,tPen\WObj:=wPaper;
    MoveL Offs(pOrigin,231.94,238.96,0.00),v40,z0,tPen\WObj:=wPaper;
    MoveL Offs(pOrigin,233.00,239.18,0.00),v40,z0,tPen\WObj:=wPaper;
    MoveL Offs(pOrigin,233.43,238.75,0.00),v40,z0,tPen\WObj:=wPaper;
    MoveL Offs(pOrigin,233.43,238.11,0.00),v40,z0,tPen\WObj:=wPaper;
    MoveL Offs(pOrigin,233.64,238.68,0.00),v40,z0,tPen\WObj:=wPaper;
    MoveL Offs(pOrigin,235.34,239.39,0.00),v40,z0,tPen\WObj:=wPaper;
    MoveL Offs(pOrigin,235.76,240.45,0.00),v40,z0,tPen\WObj:=wPaper;
    MoveL Offs(pOrigin,235.76,240.45,0.00),v40,z0,tPen\WObj:=wPaper;
    MoveL Offs(pOrigin,234.70,240.88,0.00),v40,z0,tPen\WObj:=wPaper;
    MoveL Offs(pOrigin,234.49,241.51,0.00),v40,z0,tPen\WObj:=wPaper;
    MoveL Offs(pOrigin,233.64,241.40,0.00),v40,z0,tPen\WObj:=wPaper;
    MoveL Offs(pOrigin,234.84,242.60,0.00),v40,z0,tPen\WObj:=wPaper;
    MoveL Offs(pOrigin,235.17,242.97,0.00),v40,z0,tPen\WObj:=wPaper;
    MoveL Offs(pOrigin,247.34,230.80,0.00),v40,z0,tPen\WObj:=wPaper;
    MoveL Offs(pOrigin,248.39,231.24,0.00),v40,z0,tPen\WObj:=wPaper;
    MoveL Offs(pOrigin,236.22,243.41,0.00),v40,z0,tPen\WObj:=wPaper;
    MoveL Offs(pOrigin,236.64,242.91,0.00),v40,z0,tPen\WObj:=wPaper;
    MoveL Offs(pOrigin,234.38,240.65,0.00),v40,fine,tPen\WObj:=wPaper;
    MoveL Offs(pOrigin,234.38,240.65,6.00),v60,z5,tPen\WObj:=wPaper;
    MoveL Offs(pOrigin,235.76,240.98,6.00),vTravel,z5,tPen\WObj:=wPaper;
    MoveL Offs(pOrigin,235.76,240.98,0.00),v60,z0,tPen\WObj:=wPaper;
    MoveL Offs(pOrigin,239.38,240.98,0.00),v40,z0,tPen\WObj:=wPaper;
    MoveL Offs(pOrigin,239.16,240.66,0.00),v40,z0,tPen\WObj:=wPaper;
    MoveL Offs(pOrigin,240.01,240.66,0.00),v40,z0,tPen\WObj:=wPaper;
    MoveL Offs(pOrigin,240.65,240.24,0.00),v40,z0,tPen\WObj:=wPaper;
    MoveL Offs(pOrigin,241.29,239.93,0.00),v40,z0,tPen\WObj:=wPaper;
    MoveL Offs(pOrigin,235.98,239.93,0.00),v40,z0,tPen\WObj:=wPaper;
    MoveL Offs(pOrigin,235.98,240.52,0.00),v40,z0,tPen\WObj:=wPaper;
    MoveL Offs(pOrigin,236.75,240.88,0.00),v40,z0,tPen\WObj:=wPaper;
    MoveL Offs(pOrigin,236.61,241.65,0.00),v40,z0,tPen\WObj:=wPaper;
    MoveL Offs(pOrigin,235.83,241.51,0.00),v40,z0,tPen\WObj:=wPaper;
    MoveL Offs(pOrigin,235.98,240.52,0.00),v40,z0,tPen\WObj:=wPaper;
    MoveL Offs(pOrigin,236.61,240.45,0.00),v40,z0,tPen\WObj:=wPaper;
    MoveL Offs(pOrigin,236.61,240.24,0.00),v40,z0,tPen\WObj:=wPaper;
    MoveL Offs(pOrigin,238.10,240.24,0.00),v40,z0,tPen\WObj:=wPaper;
    MoveL Offs(pOrigin,238.31,240.45,0.00),v40,z0,tPen\WObj:=wPaper;
    MoveL Offs(pOrigin,238.31,240.45,0.00),v40,z0,tPen\WObj:=wPaper;
    MoveL Offs(pOrigin,237.68,241.30,0.00),v40,z0,tPen\WObj:=wPaper;
    MoveL Offs(pOrigin,236.82,241.30,0.00),v40,z0,tPen\WObj:=wPaper;
    MoveL Offs(pOrigin,236.40,242.04,0.00),v40,z0,tPen\WObj:=wPaper;
    MoveL Offs(pOrigin,237.46,242.04,0.00),v40,fine,tPen\WObj:=wPaper;
    MoveL Offs(pOrigin,237.46,242.04,6.00),v60,z5,tPen\WObj:=wPaper;
    MoveL Offs(pOrigin,239.03,242.31,6.00),vTravel,z5,tPen\WObj:=wPaper;
    MoveL Offs(pOrigin,239.03,242.31,0.00),v60,z0,tPen\WObj:=wPaper;
    MoveL Offs(pOrigin,224.31,227.59,0.00),v40,z0,tPen\WObj:=wPaper;
    MoveL Offs(pOrigin,224.29,228.31,0.00),v40,z0,tPen\WObj:=wPaper;
    MoveL Offs(pOrigin,229.18,228.31,0.00),v40,z0,tPen\WObj:=wPaper;
    MoveL Offs(pOrigin,228.11,228.34,0.00),v40,z0,tPen\WObj:=wPaper;
    MoveL Offs(pOrigin,228.11,235.35,0.00),v40,z0,tPen\WObj:=wPaper;
    MoveL Offs(pOrigin,227.26,235.99,0.00),v40,z0,tPen\WObj:=wPaper;
    MoveL Offs(pOrigin,227.69,236.84,0.00),v40,z0,tPen\WObj:=wPaper;
    MoveL Offs(pOrigin,228.96,236.84,0.00),v40,z0,tPen\WObj:=wPaper;
    MoveL Offs(pOrigin,228.96,236.84,0.00),v40,z0,tPen\WObj:=wPaper;
    MoveL Offs(pOrigin,229.39,237.69,0.00),v40,z0,tPen\WObj:=wPaper;
    MoveL Offs(pOrigin,230.66,237.90,0.00),v40,z0,tPen\WObj:=wPaper;
    MoveL Offs(pOrigin,230.66,237.90,0.00),v40,z0,tPen\WObj:=wPaper;
    MoveL Offs(pOrigin,230.24,235.77,0.00),v40,z0,tPen\WObj:=wPaper;
  ENDPROC

  PROC DrawPart224()
    MoveL Offs(pOrigin,230.24,235.77,0.00),v40,z0,tPen\WObj:=wPaper;
    MoveL Offs(pOrigin,229.60,235.77,0.00),v40,z0,tPen\WObj:=wPaper;
    MoveL Offs(pOrigin,228.96,236.41,0.00),v40,z0,tPen\WObj:=wPaper;
    MoveL Offs(pOrigin,228.96,236.84,0.00),v40,z0,tPen\WObj:=wPaper;
    MoveL Offs(pOrigin,229.18,236.76,0.00),v40,z0,tPen\WObj:=wPaper;
    MoveL Offs(pOrigin,269.76,236.76,0.00),v40,z0,tPen\WObj:=wPaper;
    MoveL Offs(pOrigin,269.29,236.62,0.00),v40,z0,tPen\WObj:=wPaper;
    MoveL Offs(pOrigin,269.29,234.50,0.00),v40,z0,tPen\WObj:=wPaper;
    MoveL Offs(pOrigin,269.98,234.65,0.00),v40,z0,tPen\WObj:=wPaper;
    MoveL Offs(pOrigin,259.56,234.65,0.00),v40,z0,tPen\WObj:=wPaper;
    MoveL Offs(pOrigin,259.35,234.93,0.00),v40,z0,tPen\WObj:=wPaper;
    MoveL Offs(pOrigin,256.80,235.56,0.00),v40,z0,tPen\WObj:=wPaper;
    MoveL Offs(pOrigin,256.80,235.56,0.00),v40,z0,tPen\WObj:=wPaper;
    MoveL Offs(pOrigin,256.38,235.14,0.00),v40,z0,tPen\WObj:=wPaper;
    MoveL Offs(pOrigin,255.31,235.14,0.00),v40,z0,tPen\WObj:=wPaper;
    MoveL Offs(pOrigin,254.89,235.56,0.00),v40,z0,tPen\WObj:=wPaper;
    MoveL Offs(pOrigin,254.89,235.56,0.00),v40,z0,tPen\WObj:=wPaper;
    MoveL Offs(pOrigin,255.74,236.62,0.00),v40,z0,tPen\WObj:=wPaper;
    MoveL Offs(pOrigin,256.80,235.56,0.00),v40,z0,tPen\WObj:=wPaper;
    MoveL Offs(pOrigin,256.62,236.41,0.00),v40,z0,tPen\WObj:=wPaper;
    MoveL Offs(pOrigin,256.62,240.66,0.00),v40,z0,tPen\WObj:=wPaper;
    MoveL Offs(pOrigin,255.57,240.66,0.00),v40,z0,tPen\WObj:=wPaper;
    MoveL Offs(pOrigin,255.57,236.41,0.00),v40,z0,tPen\WObj:=wPaper;
    MoveL Offs(pOrigin,254.51,236.41,0.00),v40,z0,tPen\WObj:=wPaper;
    MoveL Offs(pOrigin,254.51,240.88,0.00),v40,z0,tPen\WObj:=wPaper;
    MoveL Offs(pOrigin,253.45,241.09,0.00),v40,z0,tPen\WObj:=wPaper;
    MoveL Offs(pOrigin,253.45,236.41,0.00),v40,z0,tPen\WObj:=wPaper;
    MoveL Offs(pOrigin,252.40,236.20,0.00),v40,z0,tPen\WObj:=wPaper;
    MoveL Offs(pOrigin,252.40,241.30,0.00),v40,z0,tPen\WObj:=wPaper;
    MoveL Offs(pOrigin,252.76,242.15,0.00),v40,z0,tPen\WObj:=wPaper;
    MoveL Offs(pOrigin,253.82,241.94,0.00),v40,z0,tPen\WObj:=wPaper;
    MoveL Offs(pOrigin,253.40,242.04,0.00),v40,z0,tPen\WObj:=wPaper;
    MoveL Offs(pOrigin,248.09,242.04,0.00),v40,z0,tPen\WObj:=wPaper;
    MoveL Offs(pOrigin,248.30,241.94,0.00),v40,z0,tPen\WObj:=wPaper;
    MoveL Offs(pOrigin,248.44,243.00,0.00),v40,z0,tPen\WObj:=wPaper;
    MoveL Offs(pOrigin,249.57,243.92,0.00),v40,z0,tPen\WObj:=wPaper;
    MoveL Offs(pOrigin,251.27,244.49,0.00),v40,z0,tPen\WObj:=wPaper;
    MoveL Offs(pOrigin,252.34,244.49,0.00),v40,z0,tPen\WObj:=wPaper;
    MoveL Offs(pOrigin,252.34,244.49,0.00),v40,z0,tPen\WObj:=wPaper;
    MoveL Offs(pOrigin,252.12,243.71,0.00),v40,z0,tPen\WObj:=wPaper;
    MoveL Offs(pOrigin,250.43,243.07,0.00),v40,z0,tPen\WObj:=wPaper;
    MoveL Offs(pOrigin,249.15,242.01,0.00),v40,z0,tPen\WObj:=wPaper;
    MoveL Offs(pOrigin,248.30,241.94,0.00),v40,z0,tPen\WObj:=wPaper;
    MoveL Offs(pOrigin,248.30,241.94,0.00),v40,z0,tPen\WObj:=wPaper;
    MoveL Offs(pOrigin,246.74,240.02,0.00),v40,z0,tPen\WObj:=wPaper;
    MoveL Offs(pOrigin,245.61,239.18,0.00),v40,z0,tPen\WObj:=wPaper;
    MoveL Offs(pOrigin,245.96,238.32,0.00),v40,z0,tPen\WObj:=wPaper;
    MoveL Offs(pOrigin,246.06,238.54,0.00),v40,z0,tPen\WObj:=wPaper;
    MoveL Offs(pOrigin,246.06,236.20,0.00),v40,z0,tPen\WObj:=wPaper;
    MoveL Offs(pOrigin,245.11,235.99,0.00),v40,z0,tPen\WObj:=wPaper;
    MoveL Offs(pOrigin,245.75,235.35,0.00),v40,z0,tPen\WObj:=wPaper;
    MoveL Offs(pOrigin,247.02,235.14,0.00),v40,z0,tPen\WObj:=wPaper;
    MoveL Offs(pOrigin,246.35,234.70,0.00),v40,z0,tPen\WObj:=wPaper;
    MoveL Offs(pOrigin,254.61,242.96,0.00),v40,z0,tPen\WObj:=wPaper;
    MoveL Offs(pOrigin,255.36,242.21,0.00),v40,z0,tPen\WObj:=wPaper;
    MoveL Offs(pOrigin,247.40,234.25,0.00),v40,fine,tPen\WObj:=wPaper;
    MoveL Offs(pOrigin,247.40,234.25,6.00),v60,z5,tPen\WObj:=wPaper;
    MoveL Offs(pOrigin,248.90,234.25,6.00),vTravel,z5,tPen\WObj:=wPaper;
    MoveL Offs(pOrigin,248.90,234.25,0.00),v60,z0,tPen\WObj:=wPaper;
    MoveL Offs(pOrigin,256.86,242.22,0.00),v40,fine,tPen\WObj:=wPaper;
    MoveL Offs(pOrigin,256.86,242.22,6.00),v60,z5,tPen\WObj:=wPaper;
    MoveL Offs(pOrigin,257.68,240.66,6.00),vTravel,z5,tPen\WObj:=wPaper;
    MoveL Offs(pOrigin,257.68,240.66,0.00),v60,z0,tPen\WObj:=wPaper;
    MoveL Offs(pOrigin,257.68,236.41,0.00),v40,z0,tPen\WObj:=wPaper;
    MoveL Offs(pOrigin,258.73,236.41,0.00),v40,z0,tPen\WObj:=wPaper;
    MoveL Offs(pOrigin,258.73,240.24,0.00),v40,z0,tPen\WObj:=wPaper;
    MoveL Offs(pOrigin,259.14,240.98,0.00),v40,z0,tPen\WObj:=wPaper;
    MoveL Offs(pOrigin,247.24,240.98,0.00),v40,z0,tPen\WObj:=wPaper;
    MoveL Offs(pOrigin,248.17,240.88,0.00),v40,z0,tPen\WObj:=wPaper;
    MoveL Offs(pOrigin,248.17,235.78,0.00),v40,z0,tPen\WObj:=wPaper;
    MoveL Offs(pOrigin,249.23,235.78,0.00),v40,z0,tPen\WObj:=wPaper;
    MoveL Offs(pOrigin,249.23,241.30,0.00),v40,fine,tPen\WObj:=wPaper;
    MoveL Offs(pOrigin,249.23,241.30,6.00),v60,z5,tPen\WObj:=wPaper;
    MoveL Offs(pOrigin,250.00,242.36,6.00),vTravel,z5,tPen\WObj:=wPaper;
    MoveL Offs(pOrigin,250.00,242.36,0.00),v60,z0,tPen\WObj:=wPaper;
    MoveL Offs(pOrigin,252.76,242.15,0.00),v40,z0,tPen\WObj:=wPaper;
    MoveL Offs(pOrigin,252.76,242.57,0.00),v40,z0,tPen\WObj:=wPaper;
    MoveL Offs(pOrigin,252.34,243.64,0.00),v40,z0,tPen\WObj:=wPaper;
    MoveL Offs(pOrigin,252.76,243.10,0.00),v40,z0,tPen\WObj:=wPaper;
    MoveL Offs(pOrigin,249.36,243.10,0.00),v40,fine,tPen\WObj:=wPaper;
    MoveL Offs(pOrigin,249.36,243.10,6.00),v60,z5,tPen\WObj:=wPaper;
    MoveL Offs(pOrigin,249.98,244.29,6.00),vTravel,z5,tPen\WObj:=wPaper;
    MoveL Offs(pOrigin,249.98,244.29,0.00),v60,z0,tPen\WObj:=wPaper;
    MoveL Offs(pOrigin,235.70,230.02,0.00),v40,z0,tPen\WObj:=wPaper;
    MoveL Offs(pOrigin,236.71,229.48,0.00),v40,z0,tPen\WObj:=wPaper;
    MoveL Offs(pOrigin,226.19,240.00,0.00),v40,z0,tPen\WObj:=wPaper;
    MoveL Offs(pOrigin,226.79,240.90,0.00),v40,z0,tPen\WObj:=wPaper;
    MoveL Offs(pOrigin,228.14,239.54,0.00),v40,z0,tPen\WObj:=wPaper;
    MoveL Offs(pOrigin,228.59,240.59,0.00),v40,z0,tPen\WObj:=wPaper;
    MoveL Offs(pOrigin,227.39,241.79,0.00),v40,z0,tPen\WObj:=wPaper;
    MoveL Offs(pOrigin,227.98,242.69,0.00),v40,z0,tPen\WObj:=wPaper;
    MoveL Offs(pOrigin,229.19,241.49,0.00),v40,z0,tPen\WObj:=wPaper;
    MoveL Offs(pOrigin,229.78,242.38,0.00),v40,z0,tPen\WObj:=wPaper;
    MoveL Offs(pOrigin,228.58,243.59,0.00),v40,z0,tPen\WObj:=wPaper;
    MoveL Offs(pOrigin,229.18,244.48,0.00),v40,z0,tPen\WObj:=wPaper;
    MoveL Offs(pOrigin,230.38,243.28,0.00),v40,fine,tPen\WObj:=wPaper;
    MoveL Offs(pOrigin,230.38,243.28,6.00),v60,z5,tPen\WObj:=wPaper;
    MoveL Offs(pOrigin,231.43,242.23,6.00),vTravel,z5,tPen\WObj:=wPaper;
    MoveL Offs(pOrigin,231.43,242.23,0.00),v60,z0,tPen\WObj:=wPaper;
    MoveL Offs(pOrigin,243.15,230.51,0.00),v40,z0,tPen\WObj:=wPaper;
    MoveL Offs(pOrigin,243.20,231.54,0.00),v40,z0,tPen\WObj:=wPaper;
    MoveL Offs(pOrigin,243.95,232.29,0.00),v40,fine,tPen\WObj:=wPaper;
    MoveL Offs(pOrigin,243.95,232.29,6.00),v60,z5,tPen\WObj:=wPaper;
    MoveL Offs(pOrigin,244.25,234.09,6.00),vTravel,z5,tPen\WObj:=wPaper;
    MoveL Offs(pOrigin,244.25,234.09,0.00),v60,z0,tPen\WObj:=wPaper;
    MoveL Offs(pOrigin,254.77,244.61,0.00),v40,z0,tPen\WObj:=wPaper;
    MoveL Offs(pOrigin,253.89,245.16,0.00),v40,z0,tPen\WObj:=wPaper;
    MoveL Offs(pOrigin,268.17,230.88,0.00),v40,z0,tPen\WObj:=wPaper;
    MoveL Offs(pOrigin,268.06,231.95,0.00),v40,z0,tPen\WObj:=wPaper;
    MoveL Offs(pOrigin,269.69,233.65,0.00),v40,z0,tPen\WObj:=wPaper;
    MoveL Offs(pOrigin,270.19,235.14,0.00),v40,z0,tPen\WObj:=wPaper;
    MoveL Offs(pOrigin,270.19,236.41,0.00),v40,z0,tPen\WObj:=wPaper;
    MoveL Offs(pOrigin,269.12,238.96,0.00),v40,z0,tPen\WObj:=wPaper;
    MoveL Offs(pOrigin,269.12,238.96,0.00),v40,z0,tPen\WObj:=wPaper;
    MoveL Offs(pOrigin,268.49,239.88,0.00),v40,z0,tPen\WObj:=wPaper;
    MoveL Offs(pOrigin,266.36,240.66,0.00),v40,z0,tPen\WObj:=wPaper;
    MoveL Offs(pOrigin,266.15,240.45,0.00),v40,z0,tPen\WObj:=wPaper;
    MoveL Offs(pOrigin,263.81,240.88,0.00),v40,z0,tPen\WObj:=wPaper;
    MoveL Offs(pOrigin,263.25,240.45,0.00),v40,z0,tPen\WObj:=wPaper;
    MoveL Offs(pOrigin,263.17,239.81,0.00),v40,z0,tPen\WObj:=wPaper;
  ENDPROC

  PROC DrawPart225()
    MoveL Offs(pOrigin,263.17,239.81,0.00),v40,z0,tPen\WObj:=wPaper;
    MoveL Offs(pOrigin,262.54,240.02,0.00),v40,z0,tPen\WObj:=wPaper;
    MoveL Offs(pOrigin,261.90,240.88,0.00),v40,z0,tPen\WObj:=wPaper;
    MoveL Offs(pOrigin,261.95,241.34,0.00),v40,z0,tPen\WObj:=wPaper;
    MoveL Offs(pOrigin,253.39,232.77,0.00),v40,z0,tPen\WObj:=wPaper;
    MoveL Offs(pOrigin,253.63,231.97,0.00),v40,z0,tPen\WObj:=wPaper;
    MoveL Offs(pOrigin,244.77,240.84,0.00),v40,z0,tPen\WObj:=wPaper;
    MoveL Offs(pOrigin,244.27,240.08,0.00),v40,z0,tPen\WObj:=wPaper;
    MoveL Offs(pOrigin,233.30,229.11,0.00),v40,fine,tPen\WObj:=wPaper;
    MoveL Offs(pOrigin,233.30,229.11,6.00),v60,z5,tPen\WObj:=wPaper;
    MoveL Offs(pOrigin,234.28,230.42,6.00),vTravel,z5,tPen\WObj:=wPaper;
    MoveL Offs(pOrigin,234.28,230.42,0.00),v60,z0,tPen\WObj:=wPaper;
    MoveL Offs(pOrigin,223.22,230.42,0.00),v40,z0,tPen\WObj:=wPaper;
    MoveL Offs(pOrigin,223.23,230.25,0.00),v40,z0,tPen\WObj:=wPaper;
    MoveL Offs(pOrigin,223.01,233.23,0.00),v40,z0,tPen\WObj:=wPaper;
    MoveL Offs(pOrigin,222.68,233.43,0.00),v40,z0,tPen\WObj:=wPaper;
    MoveL Offs(pOrigin,226.28,237.03,0.00),v40,fine,tPen\WObj:=wPaper;
    MoveL Offs(pOrigin,226.28,237.03,6.00),v60,z5,tPen\WObj:=wPaper;
    MoveL Offs(pOrigin,226.41,235.70,6.00),vTravel,z5,tPen\WObj:=wPaper;
    MoveL Offs(pOrigin,226.41,235.70,0.00),v60,z0,tPen\WObj:=wPaper;
    MoveL Offs(pOrigin,269.98,235.70,0.00),v40,z0,tPen\WObj:=wPaper;
    MoveL Offs(pOrigin,270.32,236.27,0.00),v40,z0,tPen\WObj:=wPaper;
    MoveL Offs(pOrigin,265.97,231.91,0.00),v40,z0,tPen\WObj:=wPaper;
    MoveL Offs(pOrigin,266.58,232.16,0.00),v40,z0,tPen\WObj:=wPaper;
    MoveL Offs(pOrigin,267.00,231.95,0.00),v40,z0,tPen\WObj:=wPaper;
    MoveL Offs(pOrigin,266.58,232.16,0.00),v40,z0,tPen\WObj:=wPaper;
    MoveL Offs(pOrigin,267.16,231.61,0.00),v40,z0,tPen\WObj:=wPaper;
    MoveL Offs(pOrigin,270.32,234.77,0.00),v40,z0,tPen\WObj:=wPaper;
    MoveL Offs(pOrigin,270.85,234.17,0.00),v40,z0,tPen\WObj:=wPaper;
    MoveL Offs(pOrigin,263.04,241.98,0.00),v40,z0,tPen\WObj:=wPaper;
    MoveL Offs(pOrigin,263.94,242.58,0.00),v40,z0,tPen\WObj:=wPaper;
    MoveL Offs(pOrigin,271.00,235.52,0.00),v40,fine,tPen\WObj:=wPaper;
    MoveL Offs(pOrigin,271.00,235.52,6.00),v60,z5,tPen\WObj:=wPaper;
    MoveL Offs(pOrigin,270.84,237.16,6.00),vTravel,z5,tPen\WObj:=wPaper;
    MoveL Offs(pOrigin,270.84,237.16,0.00),v60,z0,tPen\WObj:=wPaper;
    MoveL Offs(pOrigin,259.12,248.89,0.00),v40,fine,tPen\WObj:=wPaper;
    MoveL Offs(pOrigin,259.12,248.89,6.00),v60,z5,tPen\WObj:=wPaper;
    MoveL Offs(pOrigin,257.48,247.54,6.00),vTravel,z5,tPen\WObj:=wPaper;
    MoveL Offs(pOrigin,257.48,247.54,0.00),v60,z0,tPen\WObj:=wPaper;
    MoveL Offs(pOrigin,253.57,251.45,0.00),v40,fine,tPen\WObj:=wPaper;
    MoveL Offs(pOrigin,253.57,251.45,6.00),v60,z5,tPen\WObj:=wPaper;
    MoveL Offs(pOrigin,255.07,252.94,6.00),vTravel,z5,tPen\WObj:=wPaper;
    MoveL Offs(pOrigin,255.07,252.94,0.00),v60,z0,tPen\WObj:=wPaper;
    MoveL Offs(pOrigin,244.40,263.61,0.00),v40,z0,tPen\WObj:=wPaper;
    MoveL Offs(pOrigin,245.09,263.30,0.00),v40,z0,tPen\WObj:=wPaper;
    MoveL Offs(pOrigin,246.89,265.11,0.00),v40,z0,tPen\WObj:=wPaper;
    MoveL Offs(pOrigin,246.81,264.46,0.00),v40,z0,tPen\WObj:=wPaper;
    MoveL Offs(pOrigin,245.75,264.89,0.00),v40,fine,tPen\WObj:=wPaper;
    MoveL Offs(pOrigin,245.75,264.89,6.00),v60,z5,tPen\WObj:=wPaper;
    MoveL Offs(pOrigin,243.30,266.00,6.00),vTravel,z5,tPen\WObj:=wPaper;
    MoveL Offs(pOrigin,243.30,266.00,0.00),v60,z0,tPen\WObj:=wPaper;
    MoveL Offs(pOrigin,252.32,275.01,0.00),v40,z0,tPen\WObj:=wPaper;
    MoveL Offs(pOrigin,252.15,275.27,0.00),v40,z0,tPen\WObj:=wPaper;
    MoveL Offs(pOrigin,263.57,263.85,0.00),v40,fine,tPen\WObj:=wPaper;
    MoveL Offs(pOrigin,263.57,263.85,6.00),v60,z5,tPen\WObj:=wPaper;
    MoveL Offs(pOrigin,262.22,263.71,6.00),vTravel,z5,tPen\WObj:=wPaper;
    MoveL Offs(pOrigin,262.22,263.71,0.00),v60,z0,tPen\WObj:=wPaper;
    MoveL Offs(pOrigin,250.95,274.98,0.00),v40,z0,tPen\WObj:=wPaper;
    MoveL Offs(pOrigin,251.06,274.45,0.00),v40,z0,tPen\WObj:=wPaper;
    MoveL Offs(pOrigin,261.05,275.94,0.00),v40,fine,tPen\WObj:=wPaper;
    MoveL Offs(pOrigin,261.05,275.94,6.00),v60,z5,tPen\WObj:=wPaper;
    MoveL Offs(pOrigin,258.08,273.72,6.00),vTravel,z5,tPen\WObj:=wPaper;
    MoveL Offs(pOrigin,258.08,273.72,0.00),v60,z0,tPen\WObj:=wPaper;
    MoveL Offs(pOrigin,250.64,273.72,0.00),v40,z0,tPen\WObj:=wPaper;
    MoveL Offs(pOrigin,250.22,274.41,0.00),v40,z0,tPen\WObj:=wPaper;
    MoveL Offs(pOrigin,244.81,269.00,0.00),v40,z0,tPen\WObj:=wPaper;
    MoveL Offs(pOrigin,244.69,267.86,0.00),v40,z0,tPen\WObj:=wPaper;
    MoveL Offs(pOrigin,245.75,267.65,0.00),v40,z0,tPen\WObj:=wPaper;
    MoveL Offs(pOrigin,245.75,267.86,0.00),v40,fine,tPen\WObj:=wPaper;
    MoveL Offs(pOrigin,245.75,267.86,6.00),v60,z5,tPen\WObj:=wPaper;
    MoveL Offs(pOrigin,247.68,267.80,6.00),vTravel,z5,tPen\WObj:=wPaper;
    MoveL Offs(pOrigin,247.68,267.80,0.00),v60,z0,tPen\WObj:=wPaper;
    MoveL Offs(pOrigin,242.27,273.20,0.00),v40,fine,tPen\WObj:=wPaper;
    MoveL Offs(pOrigin,242.27,273.20,6.00),v60,z5,tPen\WObj:=wPaper;
    MoveL Offs(pOrigin,241.97,275.00,6.00),vTravel,z5,tPen\WObj:=wPaper;
    MoveL Offs(pOrigin,241.97,275.00,0.00),v60,z0,tPen\WObj:=wPaper;
    MoveL Offs(pOrigin,248.13,268.84,0.00),v40,fine,tPen\WObj:=wPaper;
    MoveL Offs(pOrigin,248.13,268.84,6.00),v60,z5,tPen\WObj:=wPaper;
    MoveL Offs(pOrigin,247.24,270.41,6.00),vTravel,z5,tPen\WObj:=wPaper;
    MoveL Offs(pOrigin,247.24,270.41,0.00),v60,z0,tPen\WObj:=wPaper;
    MoveL Offs(pOrigin,246.18,271.90,0.00),v40,z0,tPen\WObj:=wPaper;
    MoveL Offs(pOrigin,246.25,272.54,0.00),v40,z0,tPen\WObj:=wPaper;
    MoveL Offs(pOrigin,246.81,272.96,0.00),v40,z0,tPen\WObj:=wPaper;
    MoveL Offs(pOrigin,246.81,272.96,0.00),v40,z0,tPen\WObj:=wPaper;
    MoveL Offs(pOrigin,247.24,272.54,0.00),v40,z0,tPen\WObj:=wPaper;
    MoveL Offs(pOrigin,248.73,272.54,0.00),v40,fine,tPen\WObj:=wPaper;
    MoveL Offs(pOrigin,248.73,272.54,6.00),v60,z5,tPen\WObj:=wPaper;
    MoveL Offs(pOrigin,248.73,271.05,6.00),vTravel,z5,tPen\WObj:=wPaper;
    MoveL Offs(pOrigin,248.73,271.05,0.00),v60,z0,tPen\WObj:=wPaper;
    MoveL Offs(pOrigin,248.30,270.62,0.00),v40,z0,tPen\WObj:=wPaper;
    MoveL Offs(pOrigin,247.24,270.41,0.00),v40,fine,tPen\WObj:=wPaper;
    MoveL Offs(pOrigin,247.24,270.41,6.00),v60,z5,tPen\WObj:=wPaper;
    MoveL Offs(pOrigin,245.11,270.20,6.00),vTravel,z5,tPen\WObj:=wPaper;
    MoveL Offs(pOrigin,245.11,270.20,0.00),v60,z0,tPen\WObj:=wPaper;
    MoveL Offs(pOrigin,243.98,271.26,0.00),v40,z0,tPen\WObj:=wPaper;
    MoveL Offs(pOrigin,243.13,273.17,0.00),v40,z0,tPen\WObj:=wPaper;
    MoveL Offs(pOrigin,242.14,277.64,0.00),v40,fine,tPen\WObj:=wPaper;
    MoveL Offs(pOrigin,242.14,277.64,6.00),v60,z5,tPen\WObj:=wPaper;
    MoveL Offs(pOrigin,235.53,272.48,6.00),vTravel,z5,tPen\WObj:=wPaper;
    MoveL Offs(pOrigin,235.53,272.48,0.00),v60,z0,tPen\WObj:=wPaper;
    MoveL Offs(pOrigin,237.03,270.97,0.00),v40,z0,tPen\WObj:=wPaper;
    MoveL Offs(pOrigin,236.13,270.77,0.00),v40,z0,tPen\WObj:=wPaper;
    MoveL Offs(pOrigin,232.97,267.61,0.00),v40,z0,tPen\WObj:=wPaper;
    MoveL Offs(pOrigin,234.02,267.17,0.00),v40,z0,tPen\WObj:=wPaper;
    MoveL Offs(pOrigin,236.57,269.72,0.00),v40,z0,tPen\WObj:=wPaper;
    MoveL Offs(pOrigin,237.19,269.33,0.00),v40,z0,tPen\WObj:=wPaper;
    MoveL Offs(pOrigin,235.09,271.43,0.00),v40,fine,tPen\WObj:=wPaper;
    MoveL Offs(pOrigin,235.09,271.43,6.00),v60,z5,tPen\WObj:=wPaper;
    MoveL Offs(pOrigin,234.49,268.29,6.00),vTravel,z5,tPen\WObj:=wPaper;
    MoveL Offs(pOrigin,234.49,268.29,0.00),v60,z0,tPen\WObj:=wPaper;
    MoveL Offs(pOrigin,234.56,267.65,0.00),v40,z0,tPen\WObj:=wPaper;
    MoveL Offs(pOrigin,235.34,267.01,0.00),v40,z0,tPen\WObj:=wPaper;
    MoveL Offs(pOrigin,235.27,265.74,0.00),v40,z0,tPen\WObj:=wPaper;
    MoveL Offs(pOrigin,233.85,264.60,0.00),v40,z0,tPen\WObj:=wPaper;
    MoveL Offs(pOrigin,233.21,264.46,0.00),v40,z0,tPen\WObj:=wPaper;
    MoveL Offs(pOrigin,233.21,264.46,0.00),v40,z0,tPen\WObj:=wPaper;
    MoveL Offs(pOrigin,233.28,263.61,0.00),v40,z0,tPen\WObj:=wPaper;
    MoveL Offs(pOrigin,233.85,262.98,0.00),v40,z0,tPen\WObj:=wPaper;
    MoveL Offs(pOrigin,234.91,262.83,0.00),v40,z0,tPen\WObj:=wPaper;
    MoveL Offs(pOrigin,234.84,263.54,0.00),v40,z0,tPen\WObj:=wPaper;
  ENDPROC

  PROC DrawPart226()
    MoveL Offs(pOrigin,233.85,264.46,0.00),v40,z0,tPen\WObj:=wPaper;
    MoveL Offs(pOrigin,232.79,264.46,0.00),v40,z0,tPen\WObj:=wPaper;
    MoveL Offs(pOrigin,232.15,264.25,0.00),v40,z0,tPen\WObj:=wPaper;
    MoveL Offs(pOrigin,230.45,264.89,0.00),v40,z0,tPen\WObj:=wPaper;
    MoveL Offs(pOrigin,230.38,264.89,0.00),v40,z0,tPen\WObj:=wPaper;
    MoveL Offs(pOrigin,230.17,265.45,0.00),v40,z0,tPen\WObj:=wPaper;
    MoveL Offs(pOrigin,229.39,265.74,0.00),v40,z0,tPen\WObj:=wPaper;
    MoveL Offs(pOrigin,228.40,265.52,0.00),v40,z0,tPen\WObj:=wPaper;
    MoveL Offs(pOrigin,228.96,264.89,0.00),v40,z0,tPen\WObj:=wPaper;
    MoveL Offs(pOrigin,229.81,264.67,0.00),v40,z0,tPen\WObj:=wPaper;
    MoveL Offs(pOrigin,230.38,264.89,0.00),v40,fine,tPen\WObj:=wPaper;
    MoveL Offs(pOrigin,230.38,264.89,6.00),v60,z5,tPen\WObj:=wPaper;
    MoveL Offs(pOrigin,229.39,263.16,6.00),vTravel,z5,tPen\WObj:=wPaper;
    MoveL Offs(pOrigin,229.39,263.16,0.00),v60,z0,tPen\WObj:=wPaper;
    MoveL Offs(pOrigin,219.61,263.16,0.00),v40,z0,tPen\WObj:=wPaper;
    MoveL Offs(pOrigin,219.66,262.34,0.00),v40,z0,tPen\WObj:=wPaper;
    MoveL Offs(pOrigin,219.66,261.06,0.00),v40,z0,tPen\WObj:=wPaper;
    MoveL Offs(pOrigin,220.68,261.05,0.00),v40,z0,tPen\WObj:=wPaper;
    MoveL Offs(pOrigin,217.06,261.05,0.00),v40,z0,tPen\WObj:=wPaper;
    MoveL Offs(pOrigin,216.85,261.49,0.00),v40,z0,tPen\WObj:=wPaper;
    MoveL Offs(pOrigin,217.27,261.91,0.00),v40,z0,tPen\WObj:=wPaper;
    MoveL Offs(pOrigin,216.85,261.49,0.00),v40,fine,tPen\WObj:=wPaper;
    MoveL Offs(pOrigin,216.85,261.49,6.00),v60,z5,tPen\WObj:=wPaper;
    MoveL Offs(pOrigin,218.12,262.10,6.00),vTravel,z5,tPen\WObj:=wPaper;
    MoveL Offs(pOrigin,218.12,262.10,0.00),v60,z0,tPen\WObj:=wPaper;
    MoveL Offs(pOrigin,221.31,262.10,0.00),v40,fine,tPen\WObj:=wPaper;
    MoveL Offs(pOrigin,221.31,262.10,6.00),v60,z5,tPen\WObj:=wPaper;
    MoveL Offs(pOrigin,223.89,262.12,6.00),vTravel,z5,tPen\WObj:=wPaper;
    MoveL Offs(pOrigin,223.89,262.12,0.00),v60,z0,tPen\WObj:=wPaper;
    MoveL Offs(pOrigin,223.89,264.04,0.00),v40,fine,tPen\WObj:=wPaper;
    MoveL Offs(pOrigin,223.89,264.04,6.00),v60,z5,tPen\WObj:=wPaper;
    MoveL Offs(pOrigin,219.53,264.59,6.00),vTravel,z5,tPen\WObj:=wPaper;
    MoveL Offs(pOrigin,219.53,264.59,0.00),v60,z0,tPen\WObj:=wPaper;
    MoveL Offs(pOrigin,225.09,259.03,0.00),v40,z0,tPen\WObj:=wPaper;
    MoveL Offs(pOrigin,225.16,259.80,0.00),v40,z0,tPen\WObj:=wPaper;
    MoveL Offs(pOrigin,231.77,266.41,0.00),v40,z0,tPen\WObj:=wPaper;
    MoveL Offs(pOrigin,231.51,266.59,0.00),v40,z0,tPen\WObj:=wPaper;
    MoveL Offs(pOrigin,230.45,267.01,0.00),v40,z0,tPen\WObj:=wPaper;
    MoveL Offs(pOrigin,230.45,267.01,0.00),v40,z0,tPen\WObj:=wPaper;
    MoveL Offs(pOrigin,230.66,268.08,0.00),v40,fine,tPen\WObj:=wPaper;
    MoveL Offs(pOrigin,230.66,268.08,6.00),v60,z5,tPen\WObj:=wPaper;
    MoveL Offs(pOrigin,229.18,268.29,6.00),vTravel,z5,tPen\WObj:=wPaper;
    MoveL Offs(pOrigin,229.18,268.29,0.00),v60,z0,tPen\WObj:=wPaper;
    MoveL Offs(pOrigin,225.56,268.50,0.00),v40,z0,tPen\WObj:=wPaper;
    MoveL Offs(pOrigin,225.56,268.50,0.00),v40,z0,tPen\WObj:=wPaper;
    MoveL Offs(pOrigin,222.52,268.08,0.00),v40,z0,tPen\WObj:=wPaper;
    MoveL Offs(pOrigin,223.23,267.01,0.00),v40,z0,tPen\WObj:=wPaper;
    MoveL Offs(pOrigin,225.14,267.44,0.00),v40,z0,tPen\WObj:=wPaper;
    MoveL Offs(pOrigin,229.18,267.65,0.00),v40,fine,tPen\WObj:=wPaper;
    MoveL Offs(pOrigin,229.18,267.65,6.00),v60,z5,tPen\WObj:=wPaper;
    MoveL Offs(pOrigin,231.51,266.59,6.00),vTravel,z5,tPen\WObj:=wPaper;
    MoveL Offs(pOrigin,231.51,266.59,0.00),v60,z0,tPen\WObj:=wPaper;
    MoveL Offs(pOrigin,232.36,265.74,0.00),v40,z0,tPen\WObj:=wPaper;
    MoveL Offs(pOrigin,232.79,264.46,0.00),v40,fine,tPen\WObj:=wPaper;
    MoveL Offs(pOrigin,232.79,264.46,6.00),v60,z5,tPen\WObj:=wPaper;
    MoveL Offs(pOrigin,231.72,262.10,6.00),vTravel,z5,tPen\WObj:=wPaper;
    MoveL Offs(pOrigin,231.72,262.10,0.00),v60,z0,tPen\WObj:=wPaper;
    MoveL Offs(pOrigin,234.49,262.10,0.00),v40,z0,tPen\WObj:=wPaper;
    MoveL Offs(pOrigin,234.91,261.49,0.00),v40,z0,tPen\WObj:=wPaper;
    MoveL Offs(pOrigin,233.21,261.49,0.00),v40,z0,tPen\WObj:=wPaper;
    MoveL Offs(pOrigin,233.21,261.49,0.00),v40,z0,tPen\WObj:=wPaper;
    MoveL Offs(pOrigin,232.36,261.27,0.00),v40,z0,tPen\WObj:=wPaper;
    MoveL Offs(pOrigin,231.30,261.70,0.00),v40,z0,tPen\WObj:=wPaper;
    MoveL Offs(pOrigin,231.15,261.31,0.00),v40,z0,tPen\WObj:=wPaper;
    MoveL Offs(pOrigin,237.31,267.47,0.00),v40,z0,tPen\WObj:=wPaper;
    MoveL Offs(pOrigin,237.46,267.01,0.00),v40,z0,tPen\WObj:=wPaper;
    MoveL Offs(pOrigin,237.04,266.23,0.00),v40,z0,tPen\WObj:=wPaper;
    MoveL Offs(pOrigin,236.40,266.23,0.00),v40,z0,tPen\WObj:=wPaper;
    MoveL Offs(pOrigin,235.69,267.01,0.00),v40,z0,tPen\WObj:=wPaper;
    MoveL Offs(pOrigin,236.40,267.44,0.00),v40,z0,tPen\WObj:=wPaper;
    MoveL Offs(pOrigin,236.72,268.37,0.00),v40,z0,tPen\WObj:=wPaper;
    MoveL Offs(pOrigin,230.56,262.21,0.00),v40,fine,tPen\WObj:=wPaper;
    MoveL Offs(pOrigin,230.56,262.21,6.00),v60,z5,tPen\WObj:=wPaper;
    MoveL Offs(pOrigin,232.50,261.17,6.00),vTravel,z5,tPen\WObj:=wPaper;
    MoveL Offs(pOrigin,232.50,261.17,0.00),v60,z0,tPen\WObj:=wPaper;
    MoveL Offs(pOrigin,238.66,267.33,0.00),v40,z0,tPen\WObj:=wPaper;
    MoveL Offs(pOrigin,238.39,268.12,0.00),v40,z0,tPen\WObj:=wPaper;
    MoveL Offs(pOrigin,241.25,265.27,0.00),v40,z0,tPen\WObj:=wPaper;
    MoveL Offs(pOrigin,241.95,266.14,0.00),v40,z0,tPen\WObj:=wPaper;
    MoveL Offs(pOrigin,243.76,267.94,0.00),v40,fine,tPen\WObj:=wPaper;
    MoveL Offs(pOrigin,243.76,267.94,6.00),v60,z5,tPen\WObj:=wPaper;
    MoveL Offs(pOrigin,241.09,268.41,6.00),vTravel,z5,tPen\WObj:=wPaper;
    MoveL Offs(pOrigin,241.09,268.41,0.00),v60,z0,tPen\WObj:=wPaper;
    MoveL Offs(pOrigin,250.40,259.10,0.00),v40,fine,tPen\WObj:=wPaper;
    MoveL Offs(pOrigin,250.40,259.10,6.00),v60,z5,tPen\WObj:=wPaper;
    MoveL Offs(pOrigin,249.27,258.52,6.00),vTravel,z5,tPen\WObj:=wPaper;
    MoveL Offs(pOrigin,249.27,258.52,0.00),v60,z0,tPen\WObj:=wPaper;
    MoveL Offs(pOrigin,248.37,257.62,0.00),v40,z0,tPen\WObj:=wPaper;
    MoveL Offs(pOrigin,247.62,258.37,0.00),v40,z0,tPen\WObj:=wPaper;
    MoveL Offs(pOrigin,249.73,260.47,0.00),v40,fine,tPen\WObj:=wPaper;
    MoveL Offs(pOrigin,249.73,260.47,6.00),v60,z5,tPen\WObj:=wPaper;
    MoveL Offs(pOrigin,252.34,264.25,6.00),vTravel,z5,tPen\WObj:=wPaper;
    MoveL Offs(pOrigin,252.34,264.25,0.00),v60,z0,tPen\WObj:=wPaper;
    MoveL Offs(pOrigin,252.34,264.04,0.00),v40,z0,tPen\WObj:=wPaper;
    MoveL Offs(pOrigin,252.76,264.46,0.00),v40,z0,tPen\WObj:=wPaper;
    MoveL Offs(pOrigin,254.04,264.46,0.00),v40,fine,tPen\WObj:=wPaper;
    MoveL Offs(pOrigin,254.04,264.46,6.00),v60,z5,tPen\WObj:=wPaper;
    MoveL Offs(pOrigin,252.34,264.25,6.00),vTravel,z5,tPen\WObj:=wPaper;
    MoveL Offs(pOrigin,252.34,264.25,0.00),v60,z0,tPen\WObj:=wPaper;
    MoveL Offs(pOrigin,251.27,265.74,0.00),v40,fine,tPen\WObj:=wPaper;
    MoveL Offs(pOrigin,251.27,265.74,6.00),v60,z5,tPen\WObj:=wPaper;
    MoveL Offs(pOrigin,256.63,265.89,6.00),vTravel,z5,tPen\WObj:=wPaper;
    MoveL Offs(pOrigin,256.63,265.89,0.00),v60,z0,tPen\WObj:=wPaper;
    MoveL Offs(pOrigin,260.84,270.09,0.00),v40,fine,tPen\WObj:=wPaper;
    MoveL Offs(pOrigin,260.84,270.09,6.00),v60,z5,tPen\WObj:=wPaper;
    MoveL Offs(pOrigin,262.19,269.95,6.00),vTravel,z5,tPen\WObj:=wPaper;
    MoveL Offs(pOrigin,262.19,269.95,0.00),v60,z0,tPen\WObj:=wPaper;
    MoveL Offs(pOrigin,257.08,264.84,0.00),v40,fine,tPen\WObj:=wPaper;
    MoveL Offs(pOrigin,257.08,264.84,6.00),v60,z5,tPen\WObj:=wPaper;
    MoveL Offs(pOrigin,259.79,265.31,6.00),vTravel,z5,tPen\WObj:=wPaper;
    MoveL Offs(pOrigin,259.79,265.31,0.00),v60,z0,tPen\WObj:=wPaper;
    MoveL Offs(pOrigin,259.79,268.50,0.00),v40,z0,tPen\WObj:=wPaper;
    MoveL Offs(pOrigin,260.85,268.71,0.00),v40,z0,tPen\WObj:=wPaper;
    MoveL Offs(pOrigin,260.85,265.52,0.00),v40,fine,tPen\WObj:=wPaper;
    MoveL Offs(pOrigin,260.85,265.52,6.00),v60,z5,tPen\WObj:=wPaper;
    MoveL Offs(pOrigin,261.90,266.38,6.00),vTravel,z5,tPen\WObj:=wPaper;
    MoveL Offs(pOrigin,261.90,266.38,0.00),v60,z0,tPen\WObj:=wPaper;
    MoveL Offs(pOrigin,261.90,268.71,0.00),v40,fine,tPen\WObj:=wPaper;
    MoveL Offs(pOrigin,261.90,268.71,6.00),v60,z5,tPen\WObj:=wPaper;
    MoveL Offs(pOrigin,259.14,269.77,6.00),vTravel,z5,tPen\WObj:=wPaper;
  ENDPROC

  PROC DrawPart227()
    MoveL Offs(pOrigin,259.14,269.77,0.00),v60,z0,tPen\WObj:=wPaper;
    MoveL Offs(pOrigin,258.50,269.00,0.00),v40,z0,tPen\WObj:=wPaper;
    MoveL Offs(pOrigin,255.95,268.08,0.00),v40,z0,tPen\WObj:=wPaper;
    MoveL Offs(pOrigin,254.89,268.15,0.00),v40,z0,tPen\WObj:=wPaper;
    MoveL Offs(pOrigin,254.89,268.71,0.00),v40,z0,tPen\WObj:=wPaper;
    MoveL Offs(pOrigin,255.95,269.35,0.00),v40,z0,tPen\WObj:=wPaper;
    MoveL Offs(pOrigin,255.95,269.35,0.00),v40,z0,tPen\WObj:=wPaper;
    MoveL Offs(pOrigin,257.44,269.99,0.00),v40,z0,tPen\WObj:=wPaper;
    MoveL Offs(pOrigin,259.14,269.77,0.00),v40,fine,tPen\WObj:=wPaper;
    MoveL Offs(pOrigin,259.14,269.77,6.00),v60,z5,tPen\WObj:=wPaper;
    MoveL Offs(pOrigin,254.89,260.00,6.00),vTravel,z5,tPen\WObj:=wPaper;
    MoveL Offs(pOrigin,254.89,260.00,0.00),v60,z0,tPen\WObj:=wPaper;
    MoveL Offs(pOrigin,255.31,259.79,0.00),v40,z0,tPen\WObj:=wPaper;
    MoveL Offs(pOrigin,254.89,260.00,0.00),v40,fine,tPen\WObj:=wPaper;
    MoveL Offs(pOrigin,254.89,260.00,6.00),v60,z5,tPen\WObj:=wPaper;
    MoveL Offs(pOrigin,254.16,255.34,6.00),vTravel,z5,tPen\WObj:=wPaper;
    MoveL Offs(pOrigin,254.16,255.34,0.00),v60,z0,tPen\WObj:=wPaper;
    MoveL Offs(pOrigin,256.56,252.94,0.00),v40,fine,tPen\WObj:=wPaper;
    MoveL Offs(pOrigin,256.56,252.94,6.00),v60,z5,tPen\WObj:=wPaper;
    MoveL Offs(pOrigin,258.06,252.93,6.00),vTravel,z5,tPen\WObj:=wPaper;
    MoveL Offs(pOrigin,258.06,252.93,0.00),v60,z0,tPen\WObj:=wPaper;
    MoveL Offs(pOrigin,255.96,255.04,0.00),v40,fine,tPen\WObj:=wPaper;
    MoveL Offs(pOrigin,255.96,255.04,6.00),v60,z5,tPen\WObj:=wPaper;
    MoveL Offs(pOrigin,257.46,255.03,6.00),vTravel,z5,tPen\WObj:=wPaper;
    MoveL Offs(pOrigin,257.46,255.03,0.00),v60,z0,tPen\WObj:=wPaper;
    MoveL Offs(pOrigin,259.41,253.08,0.00),v40,fine,tPen\WObj:=wPaper;
    MoveL Offs(pOrigin,259.41,253.08,6.00),v60,z5,tPen\WObj:=wPaper;
    MoveL Offs(pOrigin,260.91,253.07,6.00),vTravel,z5,tPen\WObj:=wPaper;
    MoveL Offs(pOrigin,260.91,253.07,0.00),v60,z0,tPen\WObj:=wPaper;
    MoveL Offs(pOrigin,259.10,254.88,0.00),v40,fine,tPen\WObj:=wPaper;
    MoveL Offs(pOrigin,259.10,254.88,6.00),v60,z5,tPen\WObj:=wPaper;
    MoveL Offs(pOrigin,260.45,255.02,6.00),vTravel,z5,tPen\WObj:=wPaper;
    MoveL Offs(pOrigin,260.45,255.02,0.00),v60,z0,tPen\WObj:=wPaper;
    MoveL Offs(pOrigin,262.11,253.37,0.00),v40,fine,tPen\WObj:=wPaper;
    MoveL Offs(pOrigin,262.11,253.37,6.00),v60,z5,tPen\WObj:=wPaper;
    MoveL Offs(pOrigin,263.45,253.52,6.00),vTravel,z5,tPen\WObj:=wPaper;
    MoveL Offs(pOrigin,263.45,253.52,0.00),v60,z0,tPen\WObj:=wPaper;
    MoveL Offs(pOrigin,261.95,255.02,0.00),v40,fine,tPen\WObj:=wPaper;
    MoveL Offs(pOrigin,261.95,255.02,6.00),v60,z5,tPen\WObj:=wPaper;
    MoveL Offs(pOrigin,263.15,255.31,6.00),vTravel,z5,tPen\WObj:=wPaper;
    MoveL Offs(pOrigin,263.15,255.31,0.00),v60,z0,tPen\WObj:=wPaper;
    MoveL Offs(pOrigin,264.80,253.66,0.00),v40,fine,tPen\WObj:=wPaper;
    MoveL Offs(pOrigin,264.80,253.66,6.00),v60,z5,tPen\WObj:=wPaper;
    MoveL Offs(pOrigin,266.15,253.81,6.00),vTravel,z5,tPen\WObj:=wPaper;
    MoveL Offs(pOrigin,266.15,253.81,0.00),v60,z0,tPen\WObj:=wPaper;
    MoveL Offs(pOrigin,264.50,255.46,0.00),v40,fine,tPen\WObj:=wPaper;
    MoveL Offs(pOrigin,264.50,255.46,6.00),v60,z5,tPen\WObj:=wPaper;
    MoveL Offs(pOrigin,265.69,255.76,6.00),vTravel,z5,tPen\WObj:=wPaper;
    MoveL Offs(pOrigin,265.69,255.76,0.00),v60,z0,tPen\WObj:=wPaper;
    MoveL Offs(pOrigin,267.35,254.10,0.00),v40,fine,tPen\WObj:=wPaper;
    MoveL Offs(pOrigin,267.35,254.10,6.00),v60,z5,tPen\WObj:=wPaper;
    MoveL Offs(pOrigin,268.54,254.40,6.00),vTravel,z5,tPen\WObj:=wPaper;
    MoveL Offs(pOrigin,268.54,254.40,0.00),v60,z0,tPen\WObj:=wPaper;
    MoveL Offs(pOrigin,267.04,255.90,0.00),v40,z0,tPen\WObj:=wPaper;
    MoveL Offs(pOrigin,268.09,256.35,0.00),v40,z0,tPen\WObj:=wPaper;
    MoveL Offs(pOrigin,269.74,254.69,0.00),v40,fine,tPen\WObj:=wPaper;
    MoveL Offs(pOrigin,269.74,254.69,6.00),v60,z5,tPen\WObj:=wPaper;
    MoveL Offs(pOrigin,270.94,254.99,6.00),vTravel,z5,tPen\WObj:=wPaper;
    MoveL Offs(pOrigin,270.94,254.99,0.00),v60,z0,tPen\WObj:=wPaper;
    MoveL Offs(pOrigin,269.44,256.49,0.00),v40,z0,tPen\WObj:=wPaper;
    MoveL Offs(pOrigin,270.48,256.94,0.00),v40,z0,tPen\WObj:=wPaper;
    MoveL Offs(pOrigin,271.99,255.44,0.00),v40,z0,tPen\WObj:=wPaper;
    MoveL Offs(pOrigin,273.03,255.88,0.00),v40,z0,tPen\WObj:=wPaper;
    MoveL Offs(pOrigin,271.68,257.24,0.00),v40,z0,tPen\WObj:=wPaper;
    MoveL Offs(pOrigin,272.58,257.83,0.00),v40,z0,tPen\WObj:=wPaper;
    MoveL Offs(pOrigin,273.93,256.48,0.00),v40,z0,tPen\WObj:=wPaper;
    MoveL Offs(pOrigin,274.83,257.08,0.00),v40,z0,tPen\WObj:=wPaper;
    MoveL Offs(pOrigin,273.62,258.28,0.00),v40,z0,tPen\WObj:=wPaper;
    MoveL Offs(pOrigin,274.22,259.18,0.00),v40,z0,tPen\WObj:=wPaper;
    MoveL Offs(pOrigin,275.57,257.82,0.00),v40,z0,tPen\WObj:=wPaper;
    MoveL Offs(pOrigin,276.32,258.57,0.00),v40,z0,tPen\WObj:=wPaper;
    MoveL Offs(pOrigin,274.67,260.22,0.00),v40,z0,tPen\WObj:=wPaper;
    MoveL Offs(pOrigin,275.11,261.27,0.00),v40,z0,tPen\WObj:=wPaper;
    MoveL Offs(pOrigin,276.62,259.77,0.00),v40,z0,tPen\WObj:=wPaper;
    MoveL Offs(pOrigin,275.92,260.64,0.00),v40,z0,tPen\WObj:=wPaper;
    MoveL Offs(pOrigin,275.71,261.49,0.00),v40,z0,tPen\WObj:=wPaper;
    MoveL Offs(pOrigin,276.14,261.91,0.00),v40,z0,tPen\WObj:=wPaper;
    MoveL Offs(pOrigin,276.14,262.34,0.00),v40,z0,tPen\WObj:=wPaper;
    MoveL Offs(pOrigin,275.92,263.40,0.00),v40,z0,tPen\WObj:=wPaper;
    MoveL Offs(pOrigin,276.35,263.83,0.00),v40,z0,tPen\WObj:=wPaper;
    MoveL Offs(pOrigin,277.35,263.51,0.00),v40,z0,tPen\WObj:=wPaper;
    MoveL Offs(pOrigin,275.25,265.61,0.00),v40,fine,tPen\WObj:=wPaper;
    MoveL Offs(pOrigin,275.25,265.61,6.00),v60,z5,tPen\WObj:=wPaper;
    MoveL Offs(pOrigin,275.25,264.12,6.00),vTravel,z5,tPen\WObj:=wPaper;
    MoveL Offs(pOrigin,275.25,264.12,0.00),v60,z0,tPen\WObj:=wPaper;
    MoveL Offs(pOrigin,277.06,262.31,0.00),v40,fine,tPen\WObj:=wPaper;
    MoveL Offs(pOrigin,277.06,262.31,6.00),v60,z5,tPen\WObj:=wPaper;
    MoveL Offs(pOrigin,276.91,260.96,6.00),vTravel,z5,tPen\WObj:=wPaper;
    MoveL Offs(pOrigin,276.91,260.96,0.00),v60,z0,tPen\WObj:=wPaper;
    MoveL Offs(pOrigin,275.11,262.77,0.00),v40,fine,tPen\WObj:=wPaper;
    MoveL Offs(pOrigin,275.11,262.77,6.00),v60,z5,tPen\WObj:=wPaper;
    MoveL Offs(pOrigin,277.35,265.01,6.00),vTravel,z5,tPen\WObj:=wPaper;
    MoveL Offs(pOrigin,277.35,265.01,0.00),v60,z0,tPen\WObj:=wPaper;
    MoveL Offs(pOrigin,275.10,267.26,0.00),v40,fine,tPen\WObj:=wPaper;
    MoveL Offs(pOrigin,275.10,267.26,6.00),v60,z5,tPen\WObj:=wPaper;
    MoveL Offs(pOrigin,283.36,272.66,6.00),vTravel,z5,tPen\WObj:=wPaper;
    MoveL Offs(pOrigin,283.36,272.66,0.00),v60,z0,tPen\WObj:=wPaper;
    MoveL Offs(pOrigin,292.50,272.66,0.00),v40,z0,tPen\WObj:=wPaper;
    MoveL Offs(pOrigin,292.71,272.33,0.00),v40,z0,tPen\WObj:=wPaper;
    MoveL Offs(pOrigin,293.14,272.75,0.00),v40,z0,tPen\WObj:=wPaper;
    MoveL Offs(pOrigin,292.71,272.33,0.00),v40,fine,tPen\WObj:=wPaper;
    MoveL Offs(pOrigin,292.71,272.33,6.00),v60,z5,tPen\WObj:=wPaper;
    MoveL Offs(pOrigin,292.92,274.88,6.00),vTravel,z5,tPen\WObj:=wPaper;
    MoveL Offs(pOrigin,292.92,274.88,0.00),v60,z0,tPen\WObj:=wPaper;
    MoveL Offs(pOrigin,291.65,274.88,0.00),v40,z0,tPen\WObj:=wPaper;
    MoveL Offs(pOrigin,289.31,274.02,0.00),v40,z0,tPen\WObj:=wPaper;
    MoveL Offs(pOrigin,287.61,274.02,0.00),v40,z0,tPen\WObj:=wPaper;
    MoveL Offs(pOrigin,284.64,275.30,0.00),v40,z0,tPen\WObj:=wPaper;
    MoveL Offs(pOrigin,284.00,276.79,0.00),v40,z0,tPen\WObj:=wPaper;
    MoveL Offs(pOrigin,284.21,277.42,0.00),v40,fine,tPen\WObj:=wPaper;
    MoveL Offs(pOrigin,284.21,277.42,6.00),v60,z5,tPen\WObj:=wPaper;
    MoveL Offs(pOrigin,283.02,278.70,6.00),vTravel,z5,tPen\WObj:=wPaper;
    MoveL Offs(pOrigin,283.02,278.70,0.00),v60,z0,tPen\WObj:=wPaper;
    MoveL Offs(pOrigin,283.02,273.60,0.00),v40,z0,tPen\WObj:=wPaper;
    MoveL Offs(pOrigin,284.08,273.60,0.00),v40,z0,tPen\WObj:=wPaper;
    MoveL Offs(pOrigin,284.08,274.66,0.00),v40,fine,tPen\WObj:=wPaper;
    MoveL Offs(pOrigin,284.08,274.66,6.00),v60,z5,tPen\WObj:=wPaper;
    MoveL Offs(pOrigin,281.38,275.70,6.00),vTravel,z5,tPen\WObj:=wPaper;
    MoveL Offs(pOrigin,281.38,275.70,0.00),v60,z0,tPen\WObj:=wPaper;
    MoveL Offs(pOrigin,298.21,292.53,0.00),v40,fine,tPen\WObj:=wPaper;
  ENDPROC

  PROC DrawPart228()
    MoveL Offs(pOrigin,298.21,292.53,6.00),v60,z5,tPen\WObj:=wPaper;
    MoveL Offs(pOrigin,297.39,293.78,6.00),vTravel,z5,tPen\WObj:=wPaper;
    MoveL Offs(pOrigin,297.39,293.78,0.00),v60,z0,tPen\WObj:=wPaper;
    MoveL Offs(pOrigin,287.19,293.78,0.00),v40,z0,tPen\WObj:=wPaper;
    MoveL Offs(pOrigin,287.19,294.42,0.00),v40,z0,tPen\WObj:=wPaper;
    MoveL Offs(pOrigin,287.61,293.58,0.00),v40,z0,tPen\WObj:=wPaper;
    MoveL Offs(pOrigin,288.04,293.58,0.00),v40,fine,tPen\WObj:=wPaper;
    MoveL Offs(pOrigin,288.04,293.58,6.00),v60,z5,tPen\WObj:=wPaper;
    MoveL Offs(pOrigin,286.98,295.90,6.00),vTravel,z5,tPen\WObj:=wPaper;
    MoveL Offs(pOrigin,286.98,295.90,0.00),v60,z0,tPen\WObj:=wPaper;
    MoveL Offs(pOrigin,285.91,295.90,0.00),v40,fine,tPen\WObj:=wPaper;
    MoveL Offs(pOrigin,285.91,295.90,6.00),v60,z5,tPen\WObj:=wPaper;
    MoveL Offs(pOrigin,287.29,296.54,6.00),vTravel,z5,tPen\WObj:=wPaper;
    MoveL Offs(pOrigin,287.29,296.54,0.00),v60,z0,tPen\WObj:=wPaper;
    MoveL Offs(pOrigin,279.62,288.88,0.00),v40,z0,tPen\WObj:=wPaper;
    MoveL Offs(pOrigin,280.39,289.33,0.00),v40,z0,tPen\WObj:=wPaper;
    MoveL Offs(pOrigin,282.51,288.33,0.00),v40,z0,tPen\WObj:=wPaper;
    MoveL Offs(pOrigin,283.58,287.20,0.00),v40,z0,tPen\WObj:=wPaper;
    MoveL Offs(pOrigin,283.02,288.05,0.00),v40,z0,tPen\WObj:=wPaper;
    MoveL Offs(pOrigin,283.02,289.32,0.00),v40,z0,tPen\WObj:=wPaper;
    MoveL Offs(pOrigin,283.58,289.56,0.00),v40,z0,tPen\WObj:=wPaper;
    MoveL Offs(pOrigin,280.60,289.56,0.00),v40,z0,tPen\WObj:=wPaper;
    MoveL Offs(pOrigin,280.39,290.62,0.00),v40,z0,tPen\WObj:=wPaper;
    MoveL Offs(pOrigin,287.19,290.62,0.00),v40,fine,tPen\WObj:=wPaper;
    MoveL Offs(pOrigin,287.19,290.62,6.00),v60,z5,tPen\WObj:=wPaper;
    MoveL Offs(pOrigin,287.40,288.26,6.00),vTravel,z5,tPen\WObj:=wPaper;
    MoveL Offs(pOrigin,287.40,288.26,0.00),v60,z0,tPen\WObj:=wPaper;
    MoveL Offs(pOrigin,287.83,288.05,0.00),v40,z0,tPen\WObj:=wPaper;
    MoveL Offs(pOrigin,287.40,288.26,0.00),v40,z0,tPen\WObj:=wPaper;
    MoveL Offs(pOrigin,288.25,287.84,0.00),v40,z0,tPen\WObj:=wPaper;
    MoveL Offs(pOrigin,288.67,287.62,0.00),v40,z0,tPen\WObj:=wPaper;
    MoveL Offs(pOrigin,288.25,287.84,0.00),v40,z0,tPen\WObj:=wPaper;
    MoveL Offs(pOrigin,289.31,287.45,0.00),v40,z0,tPen\WObj:=wPaper;
    MoveL Offs(pOrigin,298.02,287.45,0.00),v40,z0,tPen\WObj:=wPaper;
    MoveL Offs(pOrigin,298.02,286.39,0.00),v40,z0,tPen\WObj:=wPaper;
    MoveL Offs(pOrigin,291.01,286.39,0.00),v40,fine,tPen\WObj:=wPaper;
    MoveL Offs(pOrigin,291.01,286.39,6.00),v60,z5,tPen\WObj:=wPaper;
    MoveL Offs(pOrigin,290.16,285.50,6.00),vTravel,z5,tPen\WObj:=wPaper;
    MoveL Offs(pOrigin,290.16,285.50,0.00),v60,z0,tPen\WObj:=wPaper;
    MoveL Offs(pOrigin,290.59,284.93,0.00),v40,z0,tPen\WObj:=wPaper;
    MoveL Offs(pOrigin,291.23,284.86,0.00),v40,z0,tPen\WObj:=wPaper;
    MoveL Offs(pOrigin,292.92,285.36,0.00),v40,z0,tPen\WObj:=wPaper;
    MoveL Offs(pOrigin,293.35,286.14,0.00),v40,z0,tPen\WObj:=wPaper;
    MoveL Offs(pOrigin,293.35,286.14,0.00),v40,z0,tPen\WObj:=wPaper;
    MoveL Offs(pOrigin,295.05,286.42,0.00),v40,z0,tPen\WObj:=wPaper;
    MoveL Offs(pOrigin,295.69,287.20,0.00),v40,z0,tPen\WObj:=wPaper;
    MoveL Offs(pOrigin,295.69,287.62,0.00),v40,z0,tPen\WObj:=wPaper;
    MoveL Offs(pOrigin,295.69,303.35,0.00),v40,z0,tPen\WObj:=wPaper;
    MoveL Offs(pOrigin,296.45,304.21,0.00),v40,z0,tPen\WObj:=wPaper;
    MoveL Offs(pOrigin,279.62,287.38,0.00),v40,fine,tPen\WObj:=wPaper;
    MoveL Offs(pOrigin,279.62,287.38,6.00),v60,z5,tPen\WObj:=wPaper;
    MoveL Offs(pOrigin,278.63,286.13,6.00),vTravel,z5,tPen\WObj:=wPaper;
    MoveL Offs(pOrigin,278.63,286.13,0.00),v60,z0,tPen\WObj:=wPaper;
    MoveL Offs(pOrigin,295.16,269.60,0.00),v40,z0,tPen\WObj:=wPaper;
    MoveL Offs(pOrigin,294.84,270.62,0.00),v40,z0,tPen\WObj:=wPaper;
    MoveL Offs(pOrigin,297.60,270.62,0.00),v40,fine,tPen\WObj:=wPaper;
    MoveL Offs(pOrigin,297.60,270.62,6.00),v60,z5,tPen\WObj:=wPaper;
    MoveL Offs(pOrigin,297.40,271.84,6.00),vTravel,z5,tPen\WObj:=wPaper;
    MoveL Offs(pOrigin,297.40,271.84,0.00),v60,z0,tPen\WObj:=wPaper;
    MoveL Offs(pOrigin,303.86,265.38,0.00),v40,z0,tPen\WObj:=wPaper;
    MoveL Offs(pOrigin,303.22,264.68,0.00),v40,z0,tPen\WObj:=wPaper;
    MoveL Offs(pOrigin,301.41,262.88,0.00),v40,fine,tPen\WObj:=wPaper;
    MoveL Offs(pOrigin,301.41,262.88,6.00),v60,z5,tPen\WObj:=wPaper;
    MoveL Offs(pOrigin,301.72,264.68,6.00),vTravel,z5,tPen\WObj:=wPaper;
    MoveL Offs(pOrigin,301.72,264.68,0.00),v60,z0,tPen\WObj:=wPaper;
    MoveL Offs(pOrigin,303.22,266.18,0.00),v40,z0,tPen\WObj:=wPaper;
    MoveL Offs(pOrigin,303.71,267.02,0.00),v40,z0,tPen\WObj:=wPaper;
    MoveL Offs(pOrigin,278.16,292.57,0.00),v40,z0,tPen\WObj:=wPaper;
    MoveL Offs(pOrigin,279.19,292.92,0.00),v40,z0,tPen\WObj:=wPaper;
    MoveL Offs(pOrigin,284.90,298.63,0.00),v40,z0,tPen\WObj:=wPaper;
    MoveL Offs(pOrigin,284.42,299.10,0.00),v40,z0,tPen\WObj:=wPaper;
    MoveL Offs(pOrigin,284.21,299.52,0.00),v40,z0,tPen\WObj:=wPaper;
    MoveL Offs(pOrigin,284.42,299.10,0.00),v40,z0,tPen\WObj:=wPaper;
    MoveL Offs(pOrigin,284.15,299.38,0.00),v40,z0,tPen\WObj:=wPaper;
    MoveL Offs(pOrigin,279.04,294.27,0.00),v40,z0,tPen\WObj:=wPaper;
    MoveL Offs(pOrigin,279.32,294.84,0.00),v40,z0,tPen\WObj:=wPaper;
    MoveL Offs(pOrigin,282.73,294.84,0.00),v40,fine,tPen\WObj:=wPaper;
    MoveL Offs(pOrigin,282.73,294.84,6.00),v60,z5,tPen\WObj:=wPaper;
    MoveL Offs(pOrigin,282.09,295.90,6.00),vTravel,z5,tPen\WObj:=wPaper;
    MoveL Offs(pOrigin,282.09,295.90,0.00),v60,z0,tPen\WObj:=wPaper;
    MoveL Offs(pOrigin,279.11,295.90,0.00),v40,z0,tPen\WObj:=wPaper;
    MoveL Offs(pOrigin,279.85,296.34,0.00),v40,z0,tPen\WObj:=wPaper;
    MoveL Offs(pOrigin,279.85,298.68,0.00),v40,fine,tPen\WObj:=wPaper;
    MoveL Offs(pOrigin,279.85,298.68,6.00),v60,z5,tPen\WObj:=wPaper;
    MoveL Offs(pOrigin,278.80,298.04,6.00),vTravel,z5,tPen\WObj:=wPaper;
    MoveL Offs(pOrigin,278.80,298.04,0.00),v60,z0,tPen\WObj:=wPaper;
    MoveL Offs(pOrigin,278.80,300.38,0.00),v40,z0,tPen\WObj:=wPaper;
    MoveL Offs(pOrigin,277.74,299.95,0.00),v40,z0,tPen\WObj:=wPaper;
    MoveL Offs(pOrigin,277.74,305.69,0.00),v40,fine,tPen\WObj:=wPaper;
    MoveL Offs(pOrigin,277.74,305.69,6.00),v60,z5,tPen\WObj:=wPaper;
    MoveL Offs(pOrigin,278.69,306.75,6.00),vTravel,z5,tPen\WObj:=wPaper;
    MoveL Offs(pOrigin,278.69,306.75,0.00),v60,z0,tPen\WObj:=wPaper;
    MoveL Offs(pOrigin,275.08,306.96,0.00),v40,fine,tPen\WObj:=wPaper;
    MoveL Offs(pOrigin,275.08,306.96,6.00),v60,z5,tPen\WObj:=wPaper;
    MoveL Offs(pOrigin,274.57,305.47,6.00),vTravel,z5,tPen\WObj:=wPaper;
    MoveL Offs(pOrigin,274.57,305.47,0.00),v60,z0,tPen\WObj:=wPaper;
    MoveL Offs(pOrigin,274.57,308.66,0.00),v40,z0,tPen\WObj:=wPaper;
    MoveL Offs(pOrigin,275.63,308.88,0.00),v40,z0,tPen\WObj:=wPaper;
    MoveL Offs(pOrigin,275.63,303.14,0.00),v40,z0,tPen\WObj:=wPaper;
    MoveL Offs(pOrigin,274.86,303.29,0.00),v40,z0,tPen\WObj:=wPaper;
    MoveL Offs(pOrigin,279.96,303.29,0.00),v40,z0,tPen\WObj:=wPaper;
    MoveL Offs(pOrigin,280.81,303.56,0.00),v40,z0,tPen\WObj:=wPaper;
    MoveL Offs(pOrigin,278.90,304.41,0.00),v40,z0,tPen\WObj:=wPaper;
    MoveL Offs(pOrigin,277.62,304.62,0.00),v40,z0,tPen\WObj:=wPaper;
    MoveL Offs(pOrigin,276.56,304.41,0.00),v40,z0,tPen\WObj:=wPaper;
    MoveL Offs(pOrigin,276.56,304.41,0.00),v40,z0,tPen\WObj:=wPaper;
    MoveL Offs(pOrigin,274.01,305.33,0.00),v40,z0,tPen\WObj:=wPaper;
    MoveL Offs(pOrigin,272.31,304.62,0.00),v40,z0,tPen\WObj:=wPaper;
    MoveL Offs(pOrigin,272.93,304.58,0.00),v40,z0,tPen\WObj:=wPaper;
    MoveL Offs(pOrigin,280.44,312.10,0.00),v40,fine,tPen\WObj:=wPaper;
    MoveL Offs(pOrigin,280.44,312.10,6.00),v60,z5,tPen\WObj:=wPaper;
    MoveL Offs(pOrigin,280.81,313.76,6.00),vTravel,z5,tPen\WObj:=wPaper;
    MoveL Offs(pOrigin,280.81,313.76,0.00),v60,z0,tPen\WObj:=wPaper;
    MoveL Offs(pOrigin,281.66,313.55,0.00),v40,z0,tPen\WObj:=wPaper;
    MoveL Offs(pOrigin,282.09,313.98,0.00),v40,z0,tPen\WObj:=wPaper;
    MoveL Offs(pOrigin,282.09,313.98,0.00),v40,z0,tPen\WObj:=wPaper;
    MoveL Offs(pOrigin,284.00,313.76,0.00),v40,z0,tPen\WObj:=wPaper;
    MoveL Offs(pOrigin,284.00,313.76,0.00),v40,z0,tPen\WObj:=wPaper;
    MoveL Offs(pOrigin,285.56,312.91,0.00),v40,z0,tPen\WObj:=wPaper;
    MoveL Offs(pOrigin,285.70,312.06,0.00),v40,z0,tPen\WObj:=wPaper;
  ENDPROC

  PROC DrawPart229()
    MoveL Offs(pOrigin,285.70,312.06,0.00),v40,z0,tPen\WObj:=wPaper;
    MoveL Offs(pOrigin,286.98,311.85,0.00),v40,z0,tPen\WObj:=wPaper;
    MoveL Offs(pOrigin,287.33,312.27,0.00),v40,z0,tPen\WObj:=wPaper;
    MoveL Offs(pOrigin,287.12,313.12,0.00),v40,z0,tPen\WObj:=wPaper;
    MoveL Offs(pOrigin,284.42,314.40,0.00),v40,z0,tPen\WObj:=wPaper;
    MoveL Offs(pOrigin,284.00,313.76,0.00),v40,fine,tPen\WObj:=wPaper;
    MoveL Offs(pOrigin,284.00,313.76,6.00),v60,z5,tPen\WObj:=wPaper;
    MoveL Offs(pOrigin,282.74,314.87,6.00),vTravel,z5,tPen\WObj:=wPaper;
    MoveL Offs(pOrigin,282.74,314.87,0.00),v60,z0,tPen\WObj:=wPaper;
    MoveL Offs(pOrigin,297.76,299.85,0.00),v40,fine,tPen\WObj:=wPaper;
    MoveL Offs(pOrigin,297.76,299.85,6.00),v60,z5,tPen\WObj:=wPaper;
    MoveL Offs(pOrigin,296.54,301.18,6.00),vTravel,z5,tPen\WObj:=wPaper;
    MoveL Offs(pOrigin,296.54,301.18,0.00),v60,z0,tPen\WObj:=wPaper;
    MoveL Offs(pOrigin,294.20,301.18,0.00),v40,z0,tPen\WObj:=wPaper;
    MoveL Offs(pOrigin,294.41,301.01,0.00),v40,z0,tPen\WObj:=wPaper;
    MoveL Offs(pOrigin,293.99,301.44,0.00),v40,z0,tPen\WObj:=wPaper;
    MoveL Offs(pOrigin,293.14,301.44,0.00),v40,z0,tPen\WObj:=wPaper;
    MoveL Offs(pOrigin,292.71,301.01,0.00),v40,z0,tPen\WObj:=wPaper;
    MoveL Offs(pOrigin,292.71,301.01,0.00),v40,z0,tPen\WObj:=wPaper;
    MoveL Offs(pOrigin,293.14,300.59,0.00),v40,z0,tPen\WObj:=wPaper;
    MoveL Offs(pOrigin,294.20,300.59,0.00),v40,z0,tPen\WObj:=wPaper;
    MoveL Offs(pOrigin,295.26,301.86,0.00),v40,z0,tPen\WObj:=wPaper;
    MoveL Offs(pOrigin,294.84,301.65,0.00),v40,z0,tPen\WObj:=wPaper;
    MoveL Offs(pOrigin,295.26,301.86,0.00),v40,z0,tPen\WObj:=wPaper;
    MoveL Offs(pOrigin,294.84,301.65,0.00),v40,z0,tPen\WObj:=wPaper;
    MoveL Offs(pOrigin,294.64,302.08,0.00),v40,z0,tPen\WObj:=wPaper;
    MoveL Offs(pOrigin,294.64,304.20,0.00),v40,fine,tPen\WObj:=wPaper;
    MoveL Offs(pOrigin,294.64,304.20,6.00),v60,z5,tPen\WObj:=wPaper;
    MoveL Offs(pOrigin,293.58,302.29,6.00),vTravel,z5,tPen\WObj:=wPaper;
    MoveL Offs(pOrigin,293.58,302.29,0.00),v60,z0,tPen\WObj:=wPaper;
    MoveL Offs(pOrigin,293.58,306.32,0.00),v40,z0,tPen\WObj:=wPaper;
    MoveL Offs(pOrigin,294.20,306.46,0.00),v40,z0,tPen\WObj:=wPaper;
    MoveL Offs(pOrigin,289.74,306.46,0.00),v40,z0,tPen\WObj:=wPaper;
    MoveL Offs(pOrigin,289.31,307.51,0.00),v40,z0,tPen\WObj:=wPaper;
    MoveL Offs(pOrigin,293.77,307.51,0.00),v40,z0,tPen\WObj:=wPaper;
    MoveL Offs(pOrigin,294.06,307.80,0.00),v40,z0,tPen\WObj:=wPaper;
    MoveL Offs(pOrigin,288.05,301.78,0.00),v40,z0,tPen\WObj:=wPaper;
    MoveL Offs(pOrigin,288.25,301.44,0.00),v40,z0,tPen\WObj:=wPaper;
    MoveL Offs(pOrigin,288.04,301.86,0.00),v40,z0,tPen\WObj:=wPaper;
    MoveL Offs(pOrigin,288.25,301.44,0.00),v40,z0,tPen\WObj:=wPaper;
    MoveL Offs(pOrigin,288.67,301.23,0.00),v40,z0,tPen\WObj:=wPaper;
    MoveL Offs(pOrigin,288.89,300.80,0.00),v40,z0,tPen\WObj:=wPaper;
    MoveL Offs(pOrigin,288.67,301.23,0.00),v40,z0,tPen\WObj:=wPaper;
    MoveL Offs(pOrigin,289.10,301.18,0.00),v40,z0,tPen\WObj:=wPaper;
    MoveL Offs(pOrigin,292.08,301.18,0.00),v40,z0,tPen\WObj:=wPaper;
    MoveL Offs(pOrigin,292.71,301.01,0.00),v40,z0,tPen\WObj:=wPaper;
    MoveL Offs(pOrigin,290.59,301.72,0.00),v40,z0,tPen\WObj:=wPaper;
    MoveL Offs(pOrigin,290.23,302.29,0.00),v40,z0,tPen\WObj:=wPaper;
    MoveL Offs(pOrigin,290.38,302.92,0.00),v40,z0,tPen\WObj:=wPaper;
    MoveL Offs(pOrigin,289.95,303.29,0.00),v40,z0,tPen\WObj:=wPaper;
    MoveL Offs(pOrigin,288.25,303.29,0.00),v40,z0,tPen\WObj:=wPaper;
    MoveL Offs(pOrigin,287.75,302.98,0.00),v40,z0,tPen\WObj:=wPaper;
    MoveL Offs(pOrigin,293.77,308.99,0.00),v40,z0,tPen\WObj:=wPaper;
    MoveL Offs(pOrigin,294.14,309.45,0.00),v40,z0,tPen\WObj:=wPaper;
    MoveL Offs(pOrigin,268.75,334.84,0.00),v40,fine,tPen\WObj:=wPaper;
    MoveL Offs(pOrigin,268.75,334.84,6.00),v60,z5,tPen\WObj:=wPaper;
    MoveL Offs(pOrigin,268.24,332.46,6.00),vTravel,z5,tPen\WObj:=wPaper;
    MoveL Offs(pOrigin,268.24,332.46,0.00),v60,z0,tPen\WObj:=wPaper;
    MoveL Offs(pOrigin,268.24,328.64,0.00),v40,z0,tPen\WObj:=wPaper;
    MoveL Offs(pOrigin,268.91,328.63,0.00),v40,z0,tPen\WObj:=wPaper;
    MoveL Offs(pOrigin,266.79,328.63,0.00),v40,z0,tPen\WObj:=wPaper;
    MoveL Offs(pOrigin,265.92,328.71,0.00),v40,z0,tPen\WObj:=wPaper;
    MoveL Offs(pOrigin,272.23,322.40,0.00),v40,z0,tPen\WObj:=wPaper;
    MoveL Offs(pOrigin,271.33,321.80,0.00),v40,z0,tPen\WObj:=wPaper;
    MoveL Offs(pOrigin,265.47,327.66,0.00),v40,z0,tPen\WObj:=wPaper;
    MoveL Offs(pOrigin,265.81,327.33,0.00),v40,z0,tPen\WObj:=wPaper;
    MoveL Offs(pOrigin,270.92,332.44,0.00),v40,z0,tPen\WObj:=wPaper;
    MoveL Offs(pOrigin,271.66,331.69,0.00),v40,z0,tPen\WObj:=wPaper;
    MoveL Offs(pOrigin,252.28,312.31,0.00),v40,z0,tPen\WObj:=wPaper;
    MoveL Offs(pOrigin,253.19,312.27,0.00),v40,z0,tPen\WObj:=wPaper;
    MoveL Offs(pOrigin,254.68,312.77,0.00),v40,z0,tPen\WObj:=wPaper;
    MoveL Offs(pOrigin,256.80,314.68,0.00),v40,z0,tPen\WObj:=wPaper;
    MoveL Offs(pOrigin,258.08,315.04,0.00),v40,z0,tPen\WObj:=wPaper;
    MoveL Offs(pOrigin,258.08,315.04,0.00),v40,z0,tPen\WObj:=wPaper;
    MoveL Offs(pOrigin,259.77,315.67,0.00),v40,z0,tPen\WObj:=wPaper;
    MoveL Offs(pOrigin,260.20,316.52,0.00),v40,z0,tPen\WObj:=wPaper;
    MoveL Offs(pOrigin,260.20,316.52,0.00),v40,z0,tPen\WObj:=wPaper;
    MoveL Offs(pOrigin,261.05,317.23,0.00),v40,z0,tPen\WObj:=wPaper;
    MoveL Offs(pOrigin,264.88,318.44,0.00),v40,z0,tPen\WObj:=wPaper;
    MoveL Offs(pOrigin,264.88,318.44,0.00),v40,z0,tPen\WObj:=wPaper;
    MoveL Offs(pOrigin,265.73,318.65,0.00),v40,z0,tPen\WObj:=wPaper;
    MoveL Offs(pOrigin,265.94,318.44,0.00),v40,z0,tPen\WObj:=wPaper;
    MoveL Offs(pOrigin,265.94,318.07,0.00),v40,z0,tPen\WObj:=wPaper;
    MoveL Offs(pOrigin,267.85,318.07,0.00),v40,z0,tPen\WObj:=wPaper;
    MoveL Offs(pOrigin,268.24,317.59,0.00),v40,z0,tPen\WObj:=wPaper;
    MoveL Offs(pOrigin,268.24,311.00,0.00),v40,z0,tPen\WObj:=wPaper;
    MoveL Offs(pOrigin,268.27,310.36,0.00),v40,z0,tPen\WObj:=wPaper;
    MoveL Offs(pOrigin,268.91,309.73,0.00),v40,z0,tPen\WObj:=wPaper;
    MoveL Offs(pOrigin,270.12,310.01,0.00),v40,z0,tPen\WObj:=wPaper;
    MoveL Offs(pOrigin,270.83,309.51,0.00),v40,z0,tPen\WObj:=wPaper;
    MoveL Offs(pOrigin,271.82,309.80,0.00),v40,z0,tPen\WObj:=wPaper;
    MoveL Offs(pOrigin,272.52,309.30,0.00),v40,z0,tPen\WObj:=wPaper;
    MoveL Offs(pOrigin,274.01,309.73,0.00),v40,z0,tPen\WObj:=wPaper;
    MoveL Offs(pOrigin,274.01,309.73,0.00),v40,z0,tPen\WObj:=wPaper;
    MoveL Offs(pOrigin,275.50,309.94,0.00),v40,z0,tPen\WObj:=wPaper;
    MoveL Offs(pOrigin,275.71,309.73,0.00),v40,z0,tPen\WObj:=wPaper;
    MoveL Offs(pOrigin,276.14,309.62,0.00),v40,z0,tPen\WObj:=wPaper;
    MoveL Offs(pOrigin,269.76,309.62,0.00),v40,z0,tPen\WObj:=wPaper;
    MoveL Offs(pOrigin,269.34,308.57,0.00),v40,z0,tPen\WObj:=wPaper;
    MoveL Offs(pOrigin,278.90,308.57,0.00),v40,z0,tPen\WObj:=wPaper;
    MoveL Offs(pOrigin,278.69,307.60,0.00),v40,z0,tPen\WObj:=wPaper;
    MoveL Offs(pOrigin,280.17,307.60,0.00),v40,z0,tPen\WObj:=wPaper;
    MoveL Offs(pOrigin,280.73,307.90,0.00),v40,z0,tPen\WObj:=wPaper;
    MoveL Offs(pOrigin,275.02,302.19,0.00),v40,z0,tPen\WObj:=wPaper;
    MoveL Offs(pOrigin,275.29,302.29,0.00),v40,z0,tPen\WObj:=wPaper;
    MoveL Offs(pOrigin,274.65,302.36,0.00),v40,z0,tPen\WObj:=wPaper;
    MoveL Offs(pOrigin,273.80,303.49,0.00),v40,z0,tPen\WObj:=wPaper;
    MoveL Offs(pOrigin,272.31,303.99,0.00),v40,fine,tPen\WObj:=wPaper;
    MoveL Offs(pOrigin,272.31,303.99,6.00),v60,z5,tPen\WObj:=wPaper;
    MoveL Offs(pOrigin,273.68,303.84,6.00),vTravel,z5,tPen\WObj:=wPaper;
    MoveL Offs(pOrigin,273.68,303.84,0.00),v60,z0,tPen\WObj:=wPaper;
    MoveL Offs(pOrigin,279.69,309.85,0.00),v40,z0,tPen\WObj:=wPaper;
    MoveL Offs(pOrigin,279.75,309.30,0.00),v40,z0,tPen\WObj:=wPaper;
    MoveL Offs(pOrigin,281.02,309.94,0.00),v40,z0,tPen\WObj:=wPaper;
    MoveL Offs(pOrigin,282.73,309.73,0.00),v40,fine,tPen\WObj:=wPaper;
    MoveL Offs(pOrigin,282.73,309.73,6.00),v60,z5,tPen\WObj:=wPaper;
    MoveL Offs(pOrigin,281.55,310.08,6.00),vTravel,z5,tPen\WObj:=wPaper;
    MoveL Offs(pOrigin,281.55,310.08,0.00),v60,z0,tPen\WObj:=wPaper;
    MoveL Offs(pOrigin,271.34,320.30,0.00),v40,z0,tPen\WObj:=wPaper;
    MoveL Offs(pOrigin,271.18,319.26,0.00),v40,z0,tPen\WObj:=wPaper;
  ENDPROC

  PROC DrawPart230()
    MoveL Offs(pOrigin,261.86,309.94,0.00),v40,z0,tPen\WObj:=wPaper;
    MoveL Offs(pOrigin,261.78,308.95,0.00),v40,z0,tPen\WObj:=wPaper;
    MoveL Offs(pOrigin,243.15,327.58,0.00),v40,z0,tPen\WObj:=wPaper;
    MoveL Offs(pOrigin,243.49,327.41,0.00),v40,z0,tPen\WObj:=wPaper;
    MoveL Offs(pOrigin,245.14,329.07,0.00),v40,fine,tPen\WObj:=wPaper;
    MoveL Offs(pOrigin,245.14,329.07,6.00),v60,z5,tPen\WObj:=wPaper;
    MoveL Offs(pOrigin,243.89,329.82,6.00),vTravel,z5,tPen\WObj:=wPaper;
    MoveL Offs(pOrigin,243.89,329.82,0.00),v60,z0,tPen\WObj:=wPaper;
    MoveL Offs(pOrigin,265.83,307.89,0.00),v40,fine,tPen\WObj:=wPaper;
    MoveL Offs(pOrigin,265.83,307.89,6.00),v60,z5,tPen\WObj:=wPaper;
    MoveL Offs(pOrigin,265.94,309.73,6.00),vTravel,z5,tPen\WObj:=wPaper;
    MoveL Offs(pOrigin,265.94,309.73,0.00),v60,z0,tPen\WObj:=wPaper;
    MoveL Offs(pOrigin,265.09,310.29,0.00),v40,z0,tPen\WObj:=wPaper;
    MoveL Offs(pOrigin,261.05,309.30,0.00),v40,z0,tPen\WObj:=wPaper;
    MoveL Offs(pOrigin,260.20,308.88,0.00),v40,z0,tPen\WObj:=wPaper;
    MoveL Offs(pOrigin,261.69,310.65,0.00),v40,z0,tPen\WObj:=wPaper;
    MoveL Offs(pOrigin,263.60,311.64,0.00),v40,z0,tPen\WObj:=wPaper;
    MoveL Offs(pOrigin,263.60,311.64,0.00),v40,z0,tPen\WObj:=wPaper;
    MoveL Offs(pOrigin,264.24,311.64,0.00),v40,z0,tPen\WObj:=wPaper;
    MoveL Offs(pOrigin,264.66,312.27,0.00),v40,z0,tPen\WObj:=wPaper;
    MoveL Offs(pOrigin,264.66,312.27,0.00),v40,z0,tPen\WObj:=wPaper;
    MoveL Offs(pOrigin,266.79,312.27,0.00),v40,z0,tPen\WObj:=wPaper;
    MoveL Offs(pOrigin,267.21,312.91,0.00),v40,z0,tPen\WObj:=wPaper;
    MoveL Offs(pOrigin,267.21,312.91,0.00),v40,z0,tPen\WObj:=wPaper;
    MoveL Offs(pOrigin,267.00,313.34,0.00),v40,z0,tPen\WObj:=wPaper;
    MoveL Offs(pOrigin,267.21,313.76,0.00),v40,z0,tPen\WObj:=wPaper;
    MoveL Offs(pOrigin,268.06,314.40,0.00),v40,z0,tPen\WObj:=wPaper;
    MoveL Offs(pOrigin,267.64,314.40,0.00),v40,z0,tPen\WObj:=wPaper;
    MoveL Offs(pOrigin,266.15,314.61,0.00),v40,z0,tPen\WObj:=wPaper;
    MoveL Offs(pOrigin,266.13,313.97,0.00),v40,z0,tPen\WObj:=wPaper;
    MoveL Offs(pOrigin,266.13,311.21,0.00),v40,z0,tPen\WObj:=wPaper;
    MoveL Offs(pOrigin,267.18,311.21,0.00),v40,z0,tPen\WObj:=wPaper;
    MoveL Offs(pOrigin,267.18,317.80,0.00),v40,z0,tPen\WObj:=wPaper;
    MoveL Offs(pOrigin,266.13,317.59,0.00),v40,z0,tPen\WObj:=wPaper;
    MoveL Offs(pOrigin,266.13,315.25,0.00),v40,z0,tPen\WObj:=wPaper;
    MoveL Offs(pOrigin,265.07,315.04,0.00),v40,z0,tPen\WObj:=wPaper;
    MoveL Offs(pOrigin,265.07,317.38,0.00),v40,z0,tPen\WObj:=wPaper;
    MoveL Offs(pOrigin,264.01,317.16,0.00),v40,z0,tPen\WObj:=wPaper;
    MoveL Offs(pOrigin,264.01,315.04,0.00),v40,z0,tPen\WObj:=wPaper;
    MoveL Offs(pOrigin,262.96,314.82,0.00),v40,z0,tPen\WObj:=wPaper;
    MoveL Offs(pOrigin,262.96,316.74,0.00),v40,z0,tPen\WObj:=wPaper;
    MoveL Offs(pOrigin,262.11,316.31,0.00),v40,z0,tPen\WObj:=wPaper;
    MoveL Offs(pOrigin,262.11,317.38,0.00),v40,z0,tPen\WObj:=wPaper;
    MoveL Offs(pOrigin,262.11,316.31,0.00),v40,z0,tPen\WObj:=wPaper;
    MoveL Offs(pOrigin,260.84,316.10,0.00),v40,z0,tPen\WObj:=wPaper;
    MoveL Offs(pOrigin,260.62,316.52,0.00),v40,z0,tPen\WObj:=wPaper;
    MoveL Offs(pOrigin,259.79,316.52,0.00),v40,z0,tPen\WObj:=wPaper;
    MoveL Offs(pOrigin,259.79,317.80,0.00),v40,z0,tPen\WObj:=wPaper;
    MoveL Offs(pOrigin,258.73,317.59,0.00),v40,z0,tPen\WObj:=wPaper;
    MoveL Offs(pOrigin,258.73,316.10,0.00),v40,z0,tPen\WObj:=wPaper;
    MoveL Offs(pOrigin,258.71,315.25,0.00),v40,z0,tPen\WObj:=wPaper;
    MoveL Offs(pOrigin,259.14,315.46,0.00),v40,z0,tPen\WObj:=wPaper;
    MoveL Offs(pOrigin,258.71,315.25,0.00),v40,z0,tPen\WObj:=wPaper;
    MoveL Offs(pOrigin,258.92,314.90,0.00),v40,z0,tPen\WObj:=wPaper;
    MoveL Offs(pOrigin,271.68,314.90,0.00),v40,z0,tPen\WObj:=wPaper;
    MoveL Offs(pOrigin,271.41,315.89,0.00),v40,z0,tPen\WObj:=wPaper;
    MoveL Offs(pOrigin,271.41,317.59,0.00),v40,z0,tPen\WObj:=wPaper;
    MoveL Offs(pOrigin,270.35,317.59,0.00),v40,z0,tPen\WObj:=wPaper;
    MoveL Offs(pOrigin,270.35,314.82,0.00),v40,fine,tPen\WObj:=wPaper;
    MoveL Offs(pOrigin,270.35,314.82,6.00),v60,z5,tPen\WObj:=wPaper;
    MoveL Offs(pOrigin,269.76,313.55,6.00),vTravel,z5,tPen\WObj:=wPaper;
    MoveL Offs(pOrigin,269.76,313.55,0.00),v60,z0,tPen\WObj:=wPaper;
    MoveL Offs(pOrigin,269.12,312.91,0.00),v40,z0,tPen\WObj:=wPaper;
    MoveL Offs(pOrigin,269.29,313.12,0.00),v40,z0,tPen\WObj:=wPaper;
    MoveL Offs(pOrigin,269.29,311.00,0.00),v40,z0,tPen\WObj:=wPaper;
    MoveL Offs(pOrigin,270.35,310.79,0.00),v40,z0,tPen\WObj:=wPaper;
    MoveL Offs(pOrigin,270.35,313.12,0.00),v40,z0,tPen\WObj:=wPaper;
    MoveL Offs(pOrigin,271.41,313.12,0.00),v40,z0,tPen\WObj:=wPaper;
    MoveL Offs(pOrigin,271.41,310.79,0.00),v40,z0,tPen\WObj:=wPaper;
    MoveL Offs(pOrigin,272.46,310.58,0.00),v40,z0,tPen\WObj:=wPaper;
    MoveL Offs(pOrigin,272.46,313.34,0.00),v40,fine,tPen\WObj:=wPaper;
    MoveL Offs(pOrigin,272.46,313.34,6.00),v60,z5,tPen\WObj:=wPaper;
    MoveL Offs(pOrigin,274.44,312.79,6.00),vTravel,z5,tPen\WObj:=wPaper;
    MoveL Offs(pOrigin,274.44,312.79,0.00),v60,z0,tPen\WObj:=wPaper;
    MoveL Offs(pOrigin,261.26,312.79,0.00),v40,fine,tPen\WObj:=wPaper;
    MoveL Offs(pOrigin,261.26,312.79,6.00),v60,z5,tPen\WObj:=wPaper;
    MoveL Offs(pOrigin,260.52,311.59,6.00),vTravel,z5,tPen\WObj:=wPaper;
    MoveL Offs(pOrigin,260.52,311.59,0.00),v60,z0,tPen\WObj:=wPaper;
    MoveL Offs(pOrigin,268.33,319.40,0.00),v40,z0,tPen\WObj:=wPaper;
    MoveL Offs(pOrigin,268.49,318.86,0.00),v40,z0,tPen\WObj:=wPaper;
    MoveL Offs(pOrigin,268.70,320.35,0.00),v40,z0,tPen\WObj:=wPaper;
    MoveL Offs(pOrigin,268.49,320.35,0.00),v40,z0,tPen\WObj:=wPaper;
    MoveL Offs(pOrigin,268.19,320.75,0.00),v40,z0,tPen\WObj:=wPaper;
    MoveL Offs(pOrigin,259.47,312.03,0.00),v40,z0,tPen\WObj:=wPaper;
    MoveL Offs(pOrigin,259.14,311.21,0.00),v40,z0,tPen\WObj:=wPaper;
    MoveL Offs(pOrigin,259.77,313.12,0.00),v40,fine,tPen\WObj:=wPaper;
    MoveL Offs(pOrigin,259.77,313.12,6.00),v60,z5,tPen\WObj:=wPaper;
    MoveL Offs(pOrigin,260.85,314.40,6.00),vTravel,z5,tPen\WObj:=wPaper;
    MoveL Offs(pOrigin,260.85,314.40,0.00),v60,z0,tPen\WObj:=wPaper;
    MoveL Offs(pOrigin,260.85,315.68,0.00),v40,fine,tPen\WObj:=wPaper;
    MoveL Offs(pOrigin,260.85,315.68,6.00),v60,z5,tPen\WObj:=wPaper;
    MoveL Offs(pOrigin,261.90,316.31,6.00),vTravel,z5,tPen\WObj:=wPaper;
    MoveL Offs(pOrigin,261.90,316.31,0.00),v60,z0,tPen\WObj:=wPaper;
    MoveL Offs(pOrigin,261.90,314.61,0.00),v40,fine,tPen\WObj:=wPaper;
    MoveL Offs(pOrigin,261.90,314.61,6.00),v60,z5,tPen\WObj:=wPaper;
    MoveL Offs(pOrigin,263.60,312.27,6.00),vTravel,z5,tPen\WObj:=wPaper;
    MoveL Offs(pOrigin,263.60,312.27,0.00),v60,z0,tPen\WObj:=wPaper;
    MoveL Offs(pOrigin,264.45,312.49,0.00),v40,z0,tPen\WObj:=wPaper;
    MoveL Offs(pOrigin,264.66,312.27,0.00),v40,z0,tPen\WObj:=wPaper;
    MoveL Offs(pOrigin,265.07,312.70,0.00),v40,z0,tPen\WObj:=wPaper;
    MoveL Offs(pOrigin,265.07,313.76,0.00),v40,fine,tPen\WObj:=wPaper;
    MoveL Offs(pOrigin,265.07,313.76,6.00),v60,z5,tPen\WObj:=wPaper;
    MoveL Offs(pOrigin,263.60,312.27,6.00),vTravel,z5,tPen\WObj:=wPaper;
    MoveL Offs(pOrigin,263.60,312.27,0.00),v60,z0,tPen\WObj:=wPaper;
    MoveL Offs(pOrigin,259.14,311.21,0.00),v40,z0,tPen\WObj:=wPaper;
    MoveL Offs(pOrigin,258.63,310.60,0.00),v40,z0,tPen\WObj:=wPaper;
    MoveL Offs(pOrigin,242.71,326.53,0.00),v40,z0,tPen\WObj:=wPaper;
    MoveL Offs(pOrigin,243.41,326.94,0.00),v40,z0,tPen\WObj:=wPaper;
    MoveL Offs(pOrigin,241.93,324.60,0.00),v40,z0,tPen\WObj:=wPaper;
    MoveL Offs(pOrigin,240.01,323.18,0.00),v40,z0,tPen\WObj:=wPaper;
    MoveL Offs(pOrigin,239.66,323.33,0.00),v40,z0,tPen\WObj:=wPaper;
    MoveL Offs(pOrigin,239.59,325.88,0.00),v40,z0,tPen\WObj:=wPaper;
    MoveL Offs(pOrigin,239.80,326.30,0.00),v40,z0,tPen\WObj:=wPaper;
    MoveL Offs(pOrigin,238.74,325.66,0.00),v40,z0,tPen\WObj:=wPaper;
    MoveL Offs(pOrigin,238.10,325.73,0.00),v40,z0,tPen\WObj:=wPaper;
    MoveL Offs(pOrigin,237.89,326.09,0.00),v40,z0,tPen\WObj:=wPaper;
    MoveL Offs(pOrigin,238.10,328.85,0.00),v40,z0,tPen\WObj:=wPaper;
    MoveL Offs(pOrigin,237.53,330.98,0.00),v40,z0,tPen\WObj:=wPaper;
    MoveL Offs(pOrigin,236.90,331.61,0.00),v40,z0,tPen\WObj:=wPaper;
    MoveL Offs(pOrigin,236.61,332.67,0.00),v40,z0,tPen\WObj:=wPaper;
  ENDPROC

